(* CODESYS project HVAC Example Project.project

Project tree, tasks and I/O mapping:
  Device : CODESYS Control Win V3, 3S - Smart Software Solutions GmbH, order no. 305021, version 3.5.11.30
    application Application
      libraries: Standard, * (System); HVAC Library, 1.4.0.0 (Pfaender GmbH); HVAC Types Library, 1.0.0.0 (Pfaender GmbH); HVAC Visu Library, 1.2.0.0 (Pfaender GmbH); VisuDialogs, * (System); Util, * (System)
      task HIGH (cyclic, interval t#5ms, priority 1) calls AC_CALL_HIGH_START, AC_CALL_HIGH_END
      task LOW (cyclic, interval t#20ms, priority 10) calls AC_CALL_LOW_START, AC_CALL_LOW_END
      task TrendRecordingTask (cyclic, interval 100 ms, priority 31) calls VisuTrendStorageAccess.GlobalInstances.g_TrendRecordingManager.CyclicCall
      task MainTask (cyclic, interval t#20ms, priority 1) calls PRG, Main
      task AC_RMP_Task (cyclic, interval t#20ms, priority 30) calls AC_PRG_RMP
      task AlarmManagerTask (cyclic, interval 50 ms, priority 31) calls AlarmManager.Alarm_Prg
      task VISU_TASK (cyclic, interval 100 ms, priority 31) calls VisuElems.Visu_Prg
      Trend Recording Manager
        HC_1_Trend
      Visu/
        visualisation Header_Frame
        3_Settings/
          visualisation Settings_Start
          visualisation Settings_Persistence
          visualisation Settings_MANInfo
        2_Clock Settings/
          visualisation Clock_Settings_Start
          visualisation Clock_Holiday
          visualisation Clock_Public_Holiday
          visualisation Clock_SwitchTimeS
        1_Objects/
          HC_1/
            visualisation Settings_HC_1
            visualisation Heatcurve_HC_1
            visualisation Trend_HC_1
            visualisation Clock_HC_1
            visualisation Start_HC_1
          Room_1/
            visualisation Clock_Room_1
            visualisation Start_Room_1
          visualisation Objects_Start
          AHU_1/
            visualisation Start_AHU_1
            visualisation Clock_AHU_1
        0_Alarm/
          visualisation Alarm_Start
        4_Weather/
          visualisation Weather_Start
      visualisation Start
      program Main [CFC]
      text PersistenceConfig
      AC_Std/
        function AC_InitInternal [ST]
        global variables MODULE_INFOS
        function AC_OnlineChange [ST]
        program AC_CALL_LOW_END [ST]
        program AC_CALL_LOW_START [ST]
        global variables GVL_MODULE_TREE
        program AC_CALL_HIGH_END [ST]
        program AC_CALL_HIGH_START [ST]
        global variables GVL_PersistenceManager
        function AC_Init [ST]
      Alarm Configuration
        alarm class Warning (priority 30, acknowledge REP)
        alarm group AlarmGroup
            1 [Info]: Comparison Equal, ExpressionToCompare TRUE, Expression Main.xInfoTest - "Test Alarm Class Info"
            2 [Warning]: Comparison Equal, ExpressionToCompare TRUE, Expression Main.xWarningTest - "Test Alarm Class Warning"
            3 [Error]: Comparison Equal, ExpressionToCompare TRUE, Expression PRG.HC_1.Pump.xAlarm - "Heizkreis 1: Pumpe"
            4 [Error]: Comparison Equal, ExpressionToCompare TRUE, Expression PRG.HC_1.Pump.xAlarmFb - "Heizkreis 1: Pumpe Betriebsüberwachung"
            5 [Error]: Comparison Equal, ExpressionToCompare TRUE, Expression PRG.HC_1.TS_FT_ERR - "Heizkreis 1:  Vorlauftemperaturfühler Wert gestört"
            6 [Error]: Comparison Equal, ExpressionToCompare TRUE, Expression PRG.HC_1.TS_RT_ERR - "Heizkreis 1:  Rücklauftemperaturfühler Wert gestört"
            7 [Error]: Comparison Equal, ExpressionToCompare TRUE, Expression PRG.HC_1.Valve.xAlarm - "Heizkreis 1: Ventil"
            19 [Error]: Comparison Equal, ExpressionToCompare TRUE, Expression PRG.AHU_1.Fan.xAlarm - "RLT1: Abluftventilator"
            21 [Warning]: Comparison Equal, ExpressionToCompare FALSE, Expression PRG.AHU_1.BA_AUTO - "RLT1: Anlagenschalter auf Handbetrieb"
            10 [Warning]: Comparison NotEqual, ExpressionToCompare 0, Expression PRG.HC_1.Pump.eManModeB - "Heizkreis 1: Pumpe auf Handbetrieb (Software)"
            24 [Warning]: Comparison NotEqual, ExpressionToCompare 0, Expression PRG.AHU_1.Fan_AOO - "RLT1: Ventilator auf Handbetrieb (Hardware)"
            25 [Warning]: Comparison NotEqual, ExpressionToCompare 0, Expression PRG.AHU_1.OA_Damper_AOO - "RLT1: Außenluftklappe auf Handbetrieb (Hardware)"
            16 [Warning]: Comparison NotEqual, ExpressionToCompare 0, Expression PRG.Room_1.VEN_AOO - "Room 1: Ventil auf Handbetrieb (Hardware)"
            12 [Warning]: Comparison Equal, ExpressionToCompare FALSE, Expression PRG.HC_1.BA_AUTO - "Heizkreis 1: Anlagenwahlschalter auf Handbetrieb (Software)"
            22 [Warning]: Comparison NotEqual, ExpressionToCompare 0, Expression PRG.AHU_1.Damper_OutsideAir.eManModeB - "RLT1: Außenluftklappe auf Handbetrieb (Software)"
            11 [Warning]: Comparison NotEqual, ExpressionToCompare 0, Expression PRG.HC_1.Valve.eManModeN - "Heizkreis 1: Ventil auf Handbetrieb (Software)"
            13 [Error]: Comparison Equal, ExpressionToCompare TRUE, Expression PRG.Room_1.RBG_TF_RT_STO - "Room 1: Raumtemperaturfühler Wert gestört"
            23 [Warning]: Comparison NotEqual, ExpressionToCompare 0, Expression PRG.AHU_1.Fan.eManModeB - "RLT1: Ventilator auf Handbetrieb (Software)"
            17 [Warning]: Comparison NotEqual, ExpressionToCompare 0, Expression PRG.Room_1.VEN.eManModeB - "Room 1: Ventil auf Handbetrieb (Software)"
            8 [Warning]: Comparison NotEqual, ExpressionToCompare 0, Expression PRG.HC_1.Pump_AOO - "Heizkreis 1: Pumpe auf Handbetrieb (Hardware)"
            9 [Warning]: Comparison NotEqual, ExpressionToCompare 0, Expression PRG.HC_1.Valve_AO - "Heizkreis 1: Ventil auf Handbetrieb (Hardware)"
            14 [Error]: Comparison Equal, ExpressionToCompare TRUE, Expression PRG.Room_1.FROST - "Room 1: Frostgefahr"
            15 [Warning]: Comparison Equal, ExpressionToCompare FALSE, Expression PRG.Room_1.BA_AUTO - "Room 1: Anlagenschalter Betriebsmodus auf Handbetrieb"
            20 [Warning]: Comparison Equal, ExpressionToCompare TRUE, Expression PRG.AHU_1.FilterMonitoringB.xAlarm - "RLT1: Abluftfilter Wartung notwendig"
            18 [Error]: Comparison Equal, ExpressionToCompare TRUE, Expression PRG.AHU_1.Damper_OutsideAir.xAlarm - "RLT1: Außenluftklappe Störung"
            0 [Error]: Comparison Equal, ExpressionToCompare TRUE, Expression Main.xErrorTest - "Test Alarm Class Error"
        alarm class Error (priority 10, acknowledge REP_ACK)
        text list AlarmGroup
        alarm class Info (priority 100, acknowledge REP)
        AlarmStorage
      Macros and frames/
        Room_DE/
          visualisation Zone_F_Therm_Start
          function block Zone_F_Therm [CFC]
        HeatingCircuit/
          visualisation HeatCurve4P_DN
          function block HeatingCircuit_VenA [CFC]
          visualisation HeatingCircuit_VenA_Settings
          Pump_Frames/
            visualisation Pump_Button
            visualisation Pump_Parameter_Dialog
          Valve_Frames/
            visualisation ValveAnalog_Parameter_Dialog
            visualisation ValveAnalog_Button
          visualisation HeatingCircuit_VenA
        Clock/
          visualisation Holiday
          visualisation PublicHoliday
          visualisation SwitchTimeS
        Exhaust air system/
          visualisation ExhaustAir
          function block ExhaustAir [CFC]
      program PRG [CFC]
      AC_FBs/
        function block AC_PersistenceManager_HVAC_Parameter [ST]
        function block AC_PersistenceManager_HVAC_Counter [ST]
        function block AC_PersistenceManager [ST]
      AC_RMP/
        program AC_PRG_RMP [ST]
        global variables AC_RMP
  libraries: AC_Persistence, * (3S - Smart Software Solutions GmbH)
  5ce3da45-db07-42e7-a21c-a00fff4ed8f6|C:\Users\Lukas_Pfaender\Desktop\bilder codesys\Warnung_aktiv.gif
  5ce3da45-db07-42e7-a21c-a00fff4ed8f6|C:\Users\Lukas_Pfaender\Desktop\bilder codesys\Wartung.gif
  5ce3da45-db07-42e7-a21c-a00fff4ed8f6|C:\Users\Lukas_Pfaender\Desktop\bilder codesys\Alarm_aktiv.gif
  PersistenceManager
    Kanäle (pChannels)
      HVAC_Parameter
        Datenspeicher (itfDataStorage)
        ASCIIFileStorage
      HVAC_Counter
        Datenspeicher (itfDataStorage)
        ASCIIFileStorage
  text list GlobalTextList
  AC_GENERATOR_DATA
  5ce3da45-db07-42e7-a21c-a00fff4ed8f6|C:\Users\Lukas_Pfaender\Desktop\bilder codesys\Alarm_inaktiv.gif
  GlobalImagePool
  text list System
*)

// Device/Application/AC_Std/MODULE_INFOS
//Code generated by Application Composer.
//Modifying generated code is not recommended!
{attribute 'global_init_slot' := '40000'}
{attribute 'init_on_onlchange'}

VAR_GLOBAL
	{attribute 'init_on_onlchange'}
	AC_PERSIST_PersistenceManager_INFO: AC_PERSIST.AC.ModuleInfo := (pbyModuleType := ADR('AC_PERSIST.PersistenceManager'));
	{attribute 'init_on_onlchange'}
	AC_PERSIST_PersistenceChannel_INFO: AC_PERSIST.AC.ModuleInfo := (pbyModuleType := ADR('AC_PERSIST.PersistenceChannel'));
	{attribute 'init_on_onlchange'}
	AC_PERSIST_ASCIIFileStorage_INFO: AC_PERSIST.AC.ModuleInfo := (pbyModuleType := ADR('AC_PERSIST.ASCIIFileStorage'));
END_VAR

// Device/Application/AC_Std/GVL_MODULE_TREE
//Code generated by Application Composer.
//Modifying generated code is not recommended!

VAR_GLOBAL
	Module_Tree: AC_PERSIST.AC.ModuleTree;
	aNodes: ARRAY[0..5] OF AC_PERSIST.AC.MNode;
	AC_Environment: AC_PERSIST.AC.MEnv;
END_VAR

// Device/Application/AC_Std/GVL_PersistenceManager
//Code generated by Application Composer.
//Modifying generated code is not recommended!

VAR_GLOBAL
	PersistenceManager: AC_PersistenceManager;
END_VAR

// Device/Application/AC_RMP/AC_RMP
//Code generated by Application Composer.
//Modifying generated code is not recommended!
{attribute 'global_init_slot' := '60000'}
{attribute 'init_on_onlchange'}

VAR_GLOBAL
	{attribute 'init_on_onlchange'}
	AC_RMP_Service: AC_PERSIST.AC.RMPService := (uiLocalAppID:=9744, uiNumberOfConnections:=0, pSendConnection:=0, pReceiveConnection:=0);
END_VAR

// Device/Application/AC_Std/AC_CALL_HIGH_START
//Code generated by Application Composer.
//Modifying generated code is not recommended!
PROGRAM AC_CALL_HIGH_START

//Code generated by Application Composer.
//Modifying generated code is not recommended!
PersistenceManager.CallPrioHIGHStart() ;

END_PROGRAM

// Device/Application/AC_Std/AC_CALL_HIGH_END
//Code generated by Application Composer.
//Modifying generated code is not recommended!
PROGRAM AC_CALL_HIGH_END

//Code generated by Application Composer.
//Modifying generated code is not recommended!
PersistenceManager.CallPrioHIGHEnd() ;

END_PROGRAM

// Device/Application/AC_Std/AC_CALL_LOW_START
//Code generated by Application Composer.
//Modifying generated code is not recommended!
PROGRAM AC_CALL_LOW_START

//Code generated by Application Composer.
//Modifying generated code is not recommended!
PersistenceManager.CallPrioLOWStart() ;

END_PROGRAM

// Device/Application/AC_Std/AC_CALL_LOW_END
//Code generated by Application Composer.
//Modifying generated code is not recommended!
PROGRAM AC_CALL_LOW_END

//Code generated by Application Composer.
//Modifying generated code is not recommended!
PersistenceManager.CallPrioLOWEnd() ;

END_PROGRAM

// Device/Application/PRG
PROGRAM PRG
VAR
	
	GebVar: STRING;
	HC_1: HeatingCircuit_VenA;
	HC_1_Line1 : HVAC.EditString;
	
	Room_1 : Zone_F_Therm;
	Room_Line1: HVAC.EditString;
	Clock7d1Ch_Demo: HVAC.Clock7d1Ch;
	Clock7d2Ch_Demo: HVAC.Clock7d2Ch;
	Holiday_Demo: HVAC.Holiday;
	SwitchTimeS_Demo: HVAC.SwitchTimeS;
	PublicHoliday_Demo: HVAC.PublicHoliday;

	AHU_1_Line1: HVAC.EditString;
	AHU_1: ExhaustAir;
END_VAR

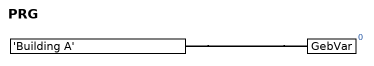
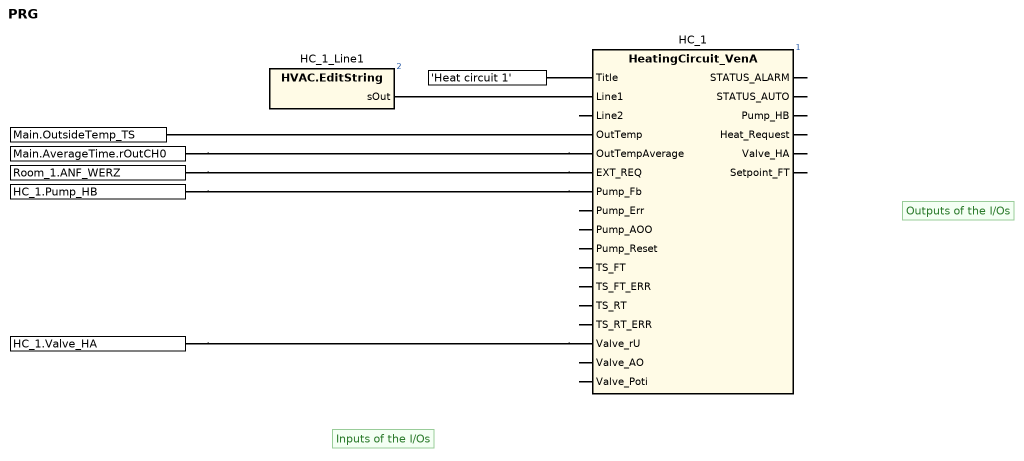
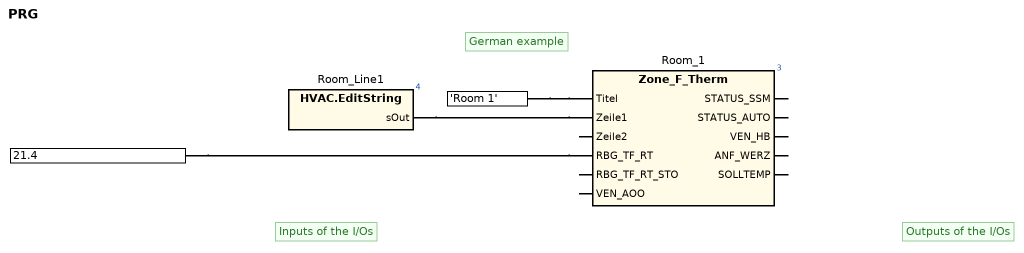
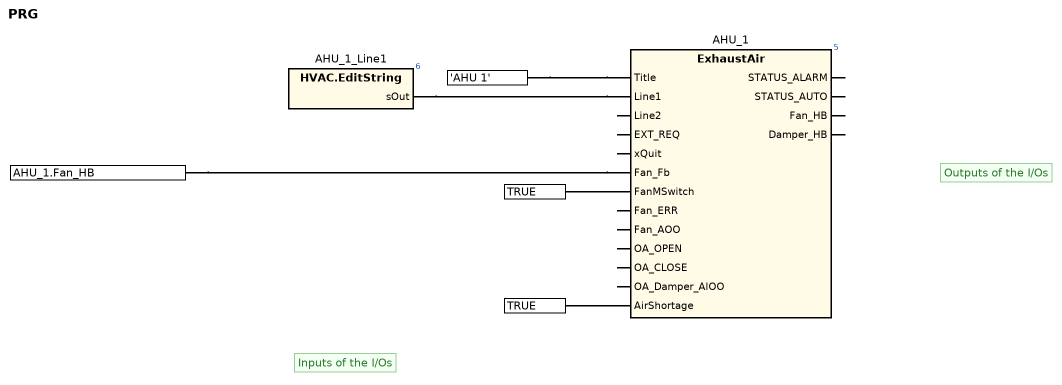
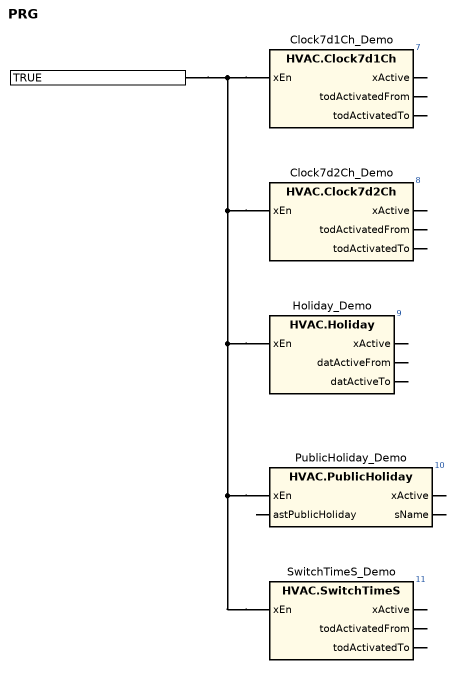
GebVar := 'Building A';
// Outputs of the I/Os
HC_1(
    Title := 'Heat circuit 1',
    Line1 := HC_1_Line1.sOut,
    OutTemp := Main.OutsideTemp_TS,
    OutTempAverage := Main.AverageTime.rOutCH0,
    EXT_REQ := Room_1.ANF_WERZ,
    Pump_Fb := HC_1.Pump_HB,
    Valve_rU := HC_1.Valve_HA); // HeatingCircuit_VenA
// Inputs of the I/Os
// parameter HC_1_Line1.sSetPoint := 'Zone 2+3'
HC_1_Line1(); // HVAC.EditString
// German example
// Outputs of the I/Os
Room_1(Titel := 'Room 1', Zeile1 := Room_Line1.sOut, RBG_TF_RT := 21.4); // Zone_F_Therm
// Inputs of the I/Os
// parameter Room_Line1.sSetPoint := 'Mr. John Doe'
Room_Line1(); // HVAC.EditString
// Outputs of the I/Os
AHU_1(
    Title := 'AHU 1',
    Line1 := AHU_1_Line1.sOut,
    Fan_Fb := AHU_1.Fan_HB,
    FanMSwitch := TRUE,
    AirShortage := TRUE); // ExhaustAir
// Inputs of the I/Os
// parameter AHU_1_Line1.sSetPoint := 'Air handling unit - exhaust air'
AHU_1_Line1(); // HVAC.EditString
Clock7d1Ch_Demo(xEn := TRUE); // HVAC.Clock7d1Ch
Clock7d2Ch_Demo(xEn := TRUE); // HVAC.Clock7d2Ch
Holiday_Demo(xEn := TRUE); // HVAC.Holiday
PublicHoliday_Demo(xEn := TRUE); // HVAC.PublicHoliday
SwitchTimeS_Demo(xEn := TRUE); // HVAC.SwitchTimeS

END_PROGRAM

// Device/Application/Main
PROGRAM Main
VAR

	TimeRead: HVAC.TimeRead;
	StartDelay: HVAC.StartDelay;
	AverageTime: HVAC.AverageTime;
	AlarmCounter: HVAC.AlarmCounter;
	Alarmgroup : UDINT := Alm_AlarmConfiguration_Alarmgroup_InternalIDs.ID_AlarmGroup;
	
	ManInfo: HVAC.ManInfo;
	ManBin_Test1: HVAC.ManBin;
	ManNum_Test1: HVAC.ManNum;
	OutsideTemp_TS: REAL := 18.5;  // Outside temperature sensor dummy. normaly analog input.

	Alarm_blink: BLINK;
	xAlarme_blinker: BOOL;
	
	xErrorTest: BOOL;
	xInfoTest  : BOOL;
	xWarningTest:BOOL;
	AlarmCounter_Warning: HVAC.AlarmCounter;
	
	OutsideTemp_TS_ERR: BOOL;						// Störung Außentemperaturfühler // Error outside temperature sensor
	checkLicense: HVAC.checkLicense;
	Outside_Temp_MAN: HVAC.ManNum;
END_VAR

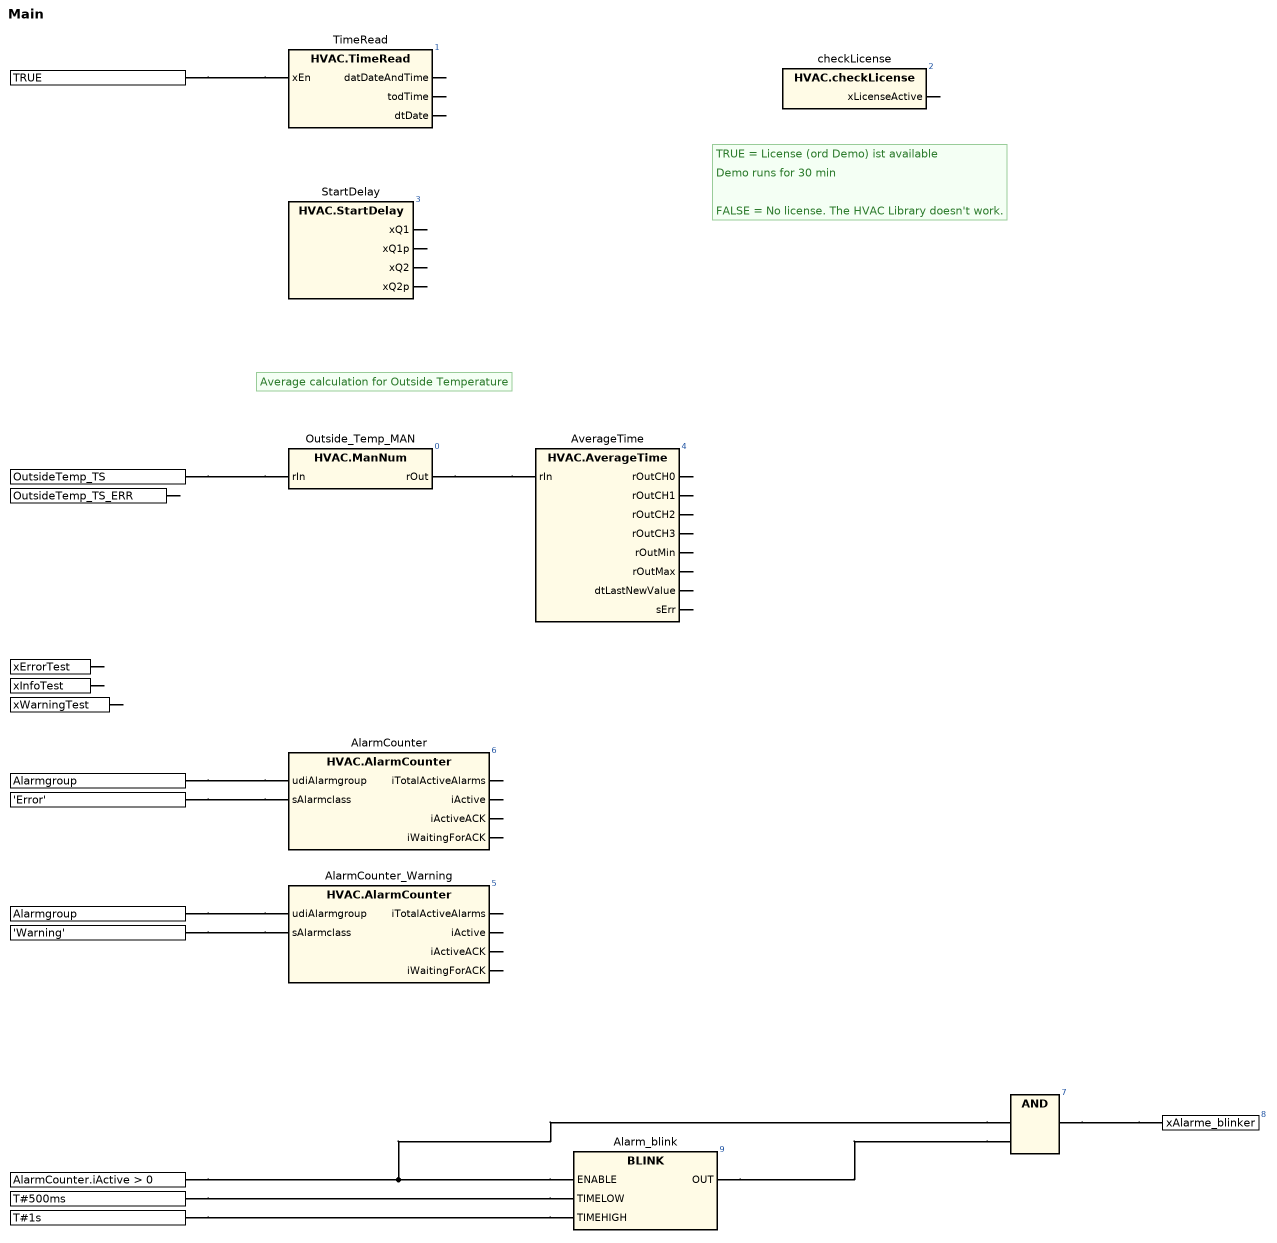
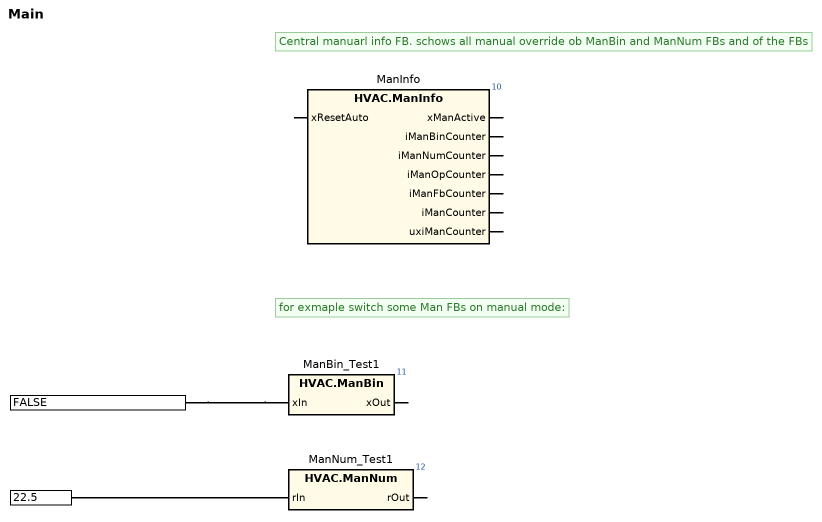
// Average calculation for Outside Temperature
Outside_Temp_MAN(rIn := OutsideTemp_TS); // HVAC.ManNum
TimeRead(xEn := TRUE); // HVAC.TimeRead
checkLicense(); // HVAC.checkLicense
// TRUE = License (ord Demo) ist available
// Demo runs for 30 min
//
// FALSE = No license. The HVAC Library doesn't work.
StartDelay(); // HVAC.StartDelay
AverageTime(rIn := Outside_Temp_MAN.rOut); // HVAC.AverageTime
AlarmCounter_Warning(udiAlarmgroup := Alarmgroup, sAlarmclass := 'Warning'); // HVAC.AlarmCounter
AlarmCounter(udiAlarmgroup := Alarmgroup, sAlarmclass := 'Error'); // HVAC.AlarmCounter
xAlarme_blinker := (AlarmCounter.iActive > 0) AND Alarm_blink.OUT;
Alarm_blink(ENABLE := AlarmCounter.iActive > 0, TIMELOW := T#500ms, TIMEHIGH := T#1s); // BLINK
// Central manuarl info FB. schows all manual override ob ManBin and ManNum FBs and of the FBs
ManInfo(); // HVAC.ManInfo
// for exmaple switch some Man FBs on manual mode:
ManBin_Test1(xIn := FALSE); // HVAC.ManBin
ManNum_Test1(rIn := 22.5); // HVAC.ManNum
// OutsideTemp_TS_ERR: input not connected
// xInfoTest: input not connected
// xWarningTest: input not connected
// xErrorTest: input not connected

END_PROGRAM

// Device/Application/Macros and frames/HeatingCircuit/HeatingCircuit_VenA
FUNCTION_BLOCK HeatingCircuit_VenA
VAR_INPUT
	Title						: STRING; 						// Name des Heizkreises  // Name of the heating circuit
	Line1						: STRING; 						// Zeile eins der Kachel // Description line 1
	Line2						: STRING; 						// Zeile zwei der Kachel // Description Line 1
	OutTemp						: REAL;							// Aussentemperaturfühler  // Outside temperature sensor
	OutTempAverage				: REAL;							// Aussentemperaturdurchschnitt // Outside temperature average
	EXT_REQ						: BOOL := FALSE;				// Externe Anforderung (Verbraucher) // External Requirement (Consumer)
	Pump_Fb						: BOOL; 						// Betrieb Umwälzpumpe // Feedback pump
	Pump_Err					: BOOL;							// Störung von Umwälzpumpe  // Alarm pump
	Pump_AOO					: HVACTypes.eManBin;			// Automatik Umwälzpumpe // pump hardware manual override(A)uto (O)ff (O)n
	Pump_Reset					: BOOL := FALSE;				// Reseteingang Störung Überwachung Betrieb  // Reset input for deedback control
	TS_FT						: REAL;							// Vorlauftemperatur // Temperature sensor flow temperature
	TS_FT_ERR					: BOOL;							// Störung Vorlauftemperaturfühler // Temperature sensor flow temperature ERROR
	TS_RT						: REAL;							// Rücklauftemperatur // Temperature sensor return temperature
	TS_RT_ERR					: BOOL;							// Störung Rücklauftemperaturfühler // Temperature sensor return temperature ERROR
	Valve_rU					: REAL;							// Rückführung Ventil  // Return Valve
	Valve_AO					: HVACTypes.eManNum;							// Automatik Ventil  //  Valve hardware manual override (A)uto (On)
	Valve_Poti					: REAL;							// Analogübersteuerung Poti // manual override potentiometer value
END_VAR

VAR_OUTPUT
	STATUS_ALARM					: BOOL;							// Sammelstörmeldung // Central Fault (Error)
	STATUS_AUTO					: BOOL;							// Statusmeldung: 0=Hand 1=Auto // Central Automatic message FALSE = manual TRUE = Auto
	Pump_HB						: BOOL;							// Ausgang Umwälzpumpe  // Output pump binary
	Heat_Request				: BOOL;							// Anforderung Wärmeerzeugung  // Heat request
	Valve_HA					: REAL;							// Ausgang Ventil // Output valve analog
	Setpoint_FT					: REAL;							// Vorlaufsolltemperatur  // Setpoint flow temperature
END_VAR
VAR
	OS							: hvac.OpModeSelect;			// Anlagen Wahlschalter // Operation mode Select
	BA_AUTO						: BOOL;							// Betriebsart Auto // Operation mode automatic
	BA_HAND0					: BOOL;							// Betriebsart HAND - Nachtbetrieb  // Operation mode: manual - night operation
	BA_HAND1					: BOOL;							// Betriebsart HAND - Tagbetrieb // Operation mode: manual - day operation
	R_OutTemp					: BOOL;							// Freigabe über Aussentemperatur  // Release via outside temperature
	R_OutTemp_MAN				: hvac.ManBin;					// Manuell Baustein für die Freigabe der Außentemperatur  // Manual function block for outside temperature release
	R_OutTemp_SR				: SR;							// Flipflop Freigabe Heizbetrieb  // Release flipflop for heating operation
	R_OutTemp_TON				: TON;							
	R_OutTemp_TOF				: TOF;
	HEAT						: BOOL;							// Heizbetrieb  // Heating operation
	HC							: hvac.HeatCurve4P_DN;			// Heizkurve // haeting curve
	MODE						: BOOL;							// Modus: FALSE=Nachtbetrieb TRUE=Tagbetrieb // Mode: FALSE=night operation TRUE=day operation
	Reg2P_HZ_AKT				: hvac.Control2P;				// Zweipunktregler Heizen aktuell  // Control two point heating mode actual
	Reg2P_HZ_DURCH				: hvac.Control2P;				// Zweipunktregler Heizen Durchschnitt //  Control two point heating mode average
	Reg2P_WINTER				: hvac.Control2P;				// Zweipunktregler Heizen Wintermodus // Control two point heating operation winter
	ConPI_FT					: hvac.ControlPI;				// PI Regler für Vorlauftemperaturregelung	// Control PI for flow temperature regulation
	Setpoint_FT_MAN				: hvac.ManNum;					// Handübersteuerung Soll Vorlauftemperatur // Manual override for setpoint flow temperature
	Setpoint_Heat_Aver				: hvac.Edit;					// Sollwert: Freigabe Heizbetrieb bei AT-Durch < // Setpoint: Release heating operation at outside temperature average <
	Setpoint_Heat_Act			: hvac.Edit;					// Sollwert: Freigabe Heizbetrieb bei Aussentemperatur < // Setpoint: Release heating operation at actual outside temperature <
	Setpoint_WINTER				: hvac.Edit;					// Sollwert: Freigabe Winterbetrieb bei AT-Durch < // Setpoint release winter operation at outside temperature average <
	STATUS_ERR_MAN				: hvac.ManBin;					// Handübersteuerung Sammelstörmeldung  // Manual override central error
	STATUS_AUTO_MAN				: hvac.ManBin;					// Handübersteuerung Automatikmeldung // Manual override central automatic notification
	Clock						: HVAC.Clock7d1Ch;				// Einkanal Wochenuhr  // One channel week clock
	Pump						: hvac.Pump;					// Umwälzpumpe  // Circuit  pump
	Clock_Channel				: BOOL;							// Uhrkanal // Clock Channel
	Valve_ERR					: BOOL;							// Störung Ventil //Valve Alarm
	WINTER						: BOOL;							// Winterbetrieb //Winter operation
	Valve						: hvac.ValveAnalog;
END_VAR
VAR // added by the converter: edge detectors and wires of the graphical bodies
    _w1, _w2, _w3, _w4, _w5, _w6, _w7 : ANY;
END_VAR

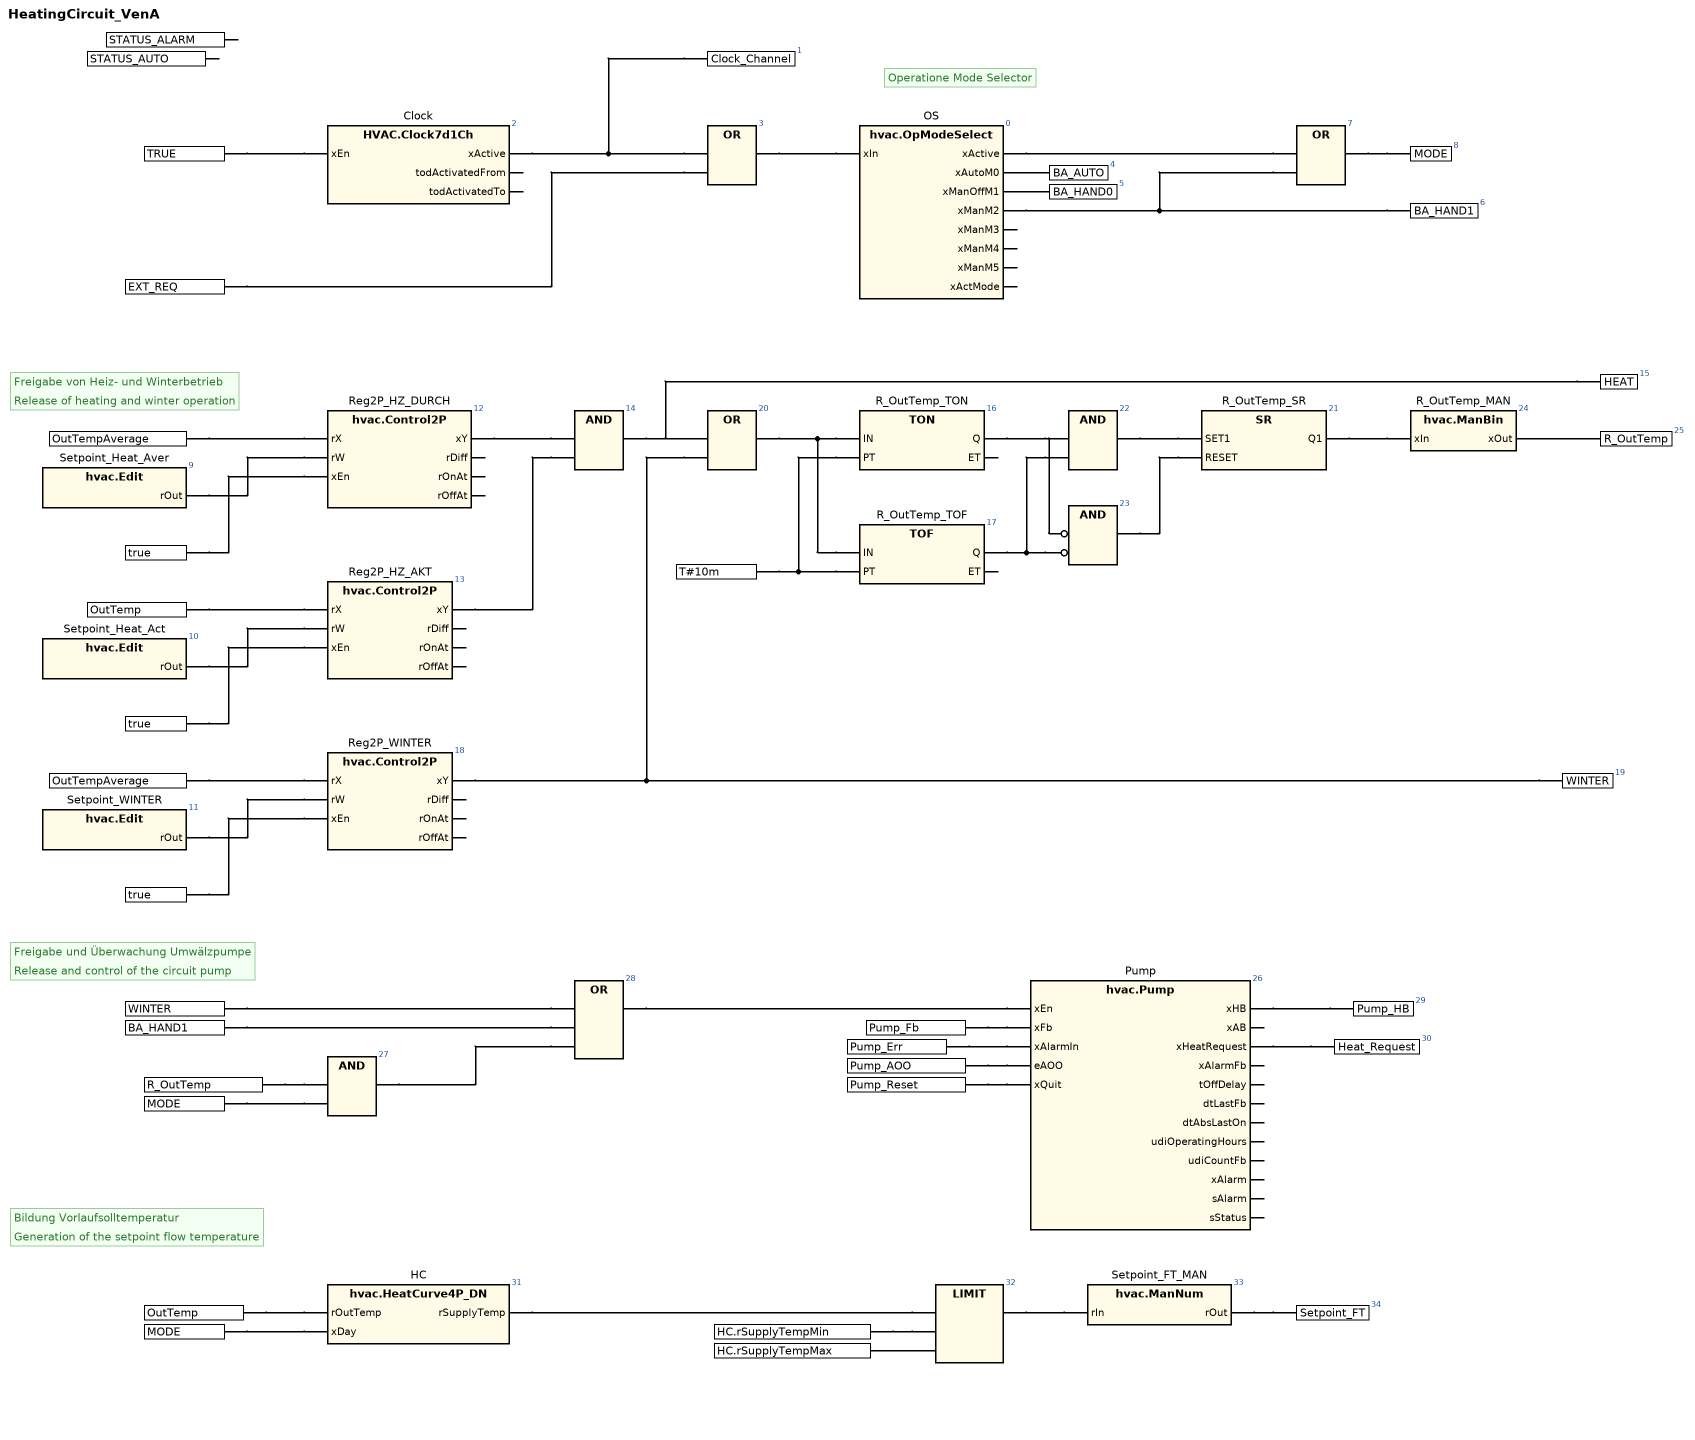
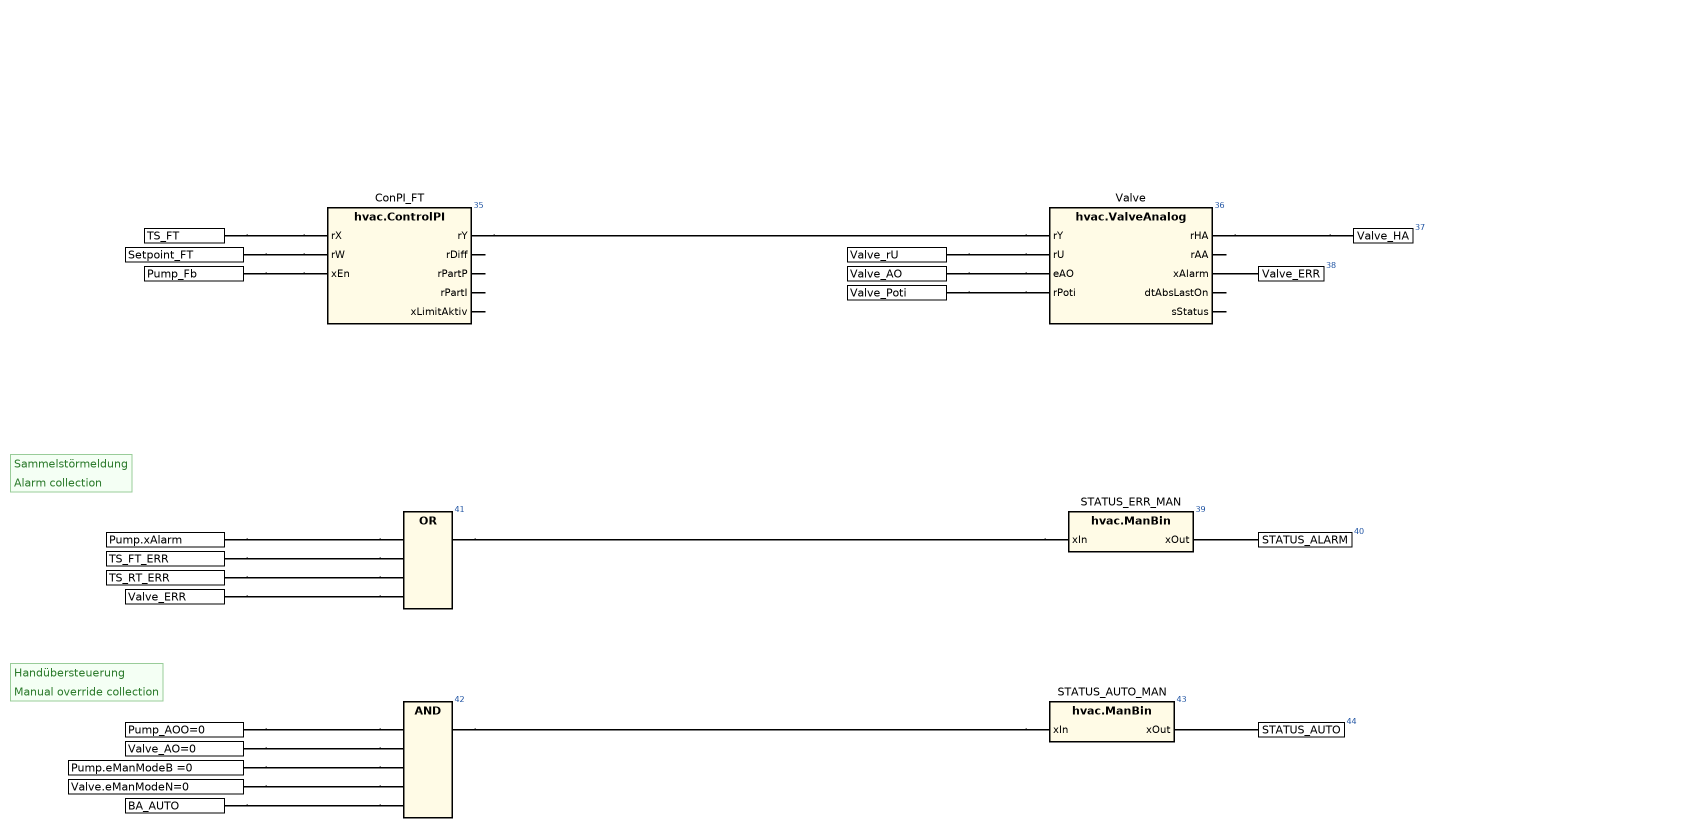
// note: 115 stored wires end on pins the file does not list and are not shown
// Operatione Mode Selector
// parameter OS.sTitleM2 := 'Manual On'
// parameter OS.sTitleM1 := 'Manual Off'
// parameter OS.sTitleM0 := 'Automatic'
// parameter OS.sTitle := 'Operation Mode'
// parameter OS.eMaxMode := HVAC.eOpMode.Mode2
OS(xIn := _w1); // hvac.OpModeSelect
Clock_Channel := Clock.xActive;
// parameter Clock.todSunTo := tod#00:00:00
// parameter Clock.todSunFrom := tod#00:00:00
// parameter Clock.todFriTo := tod#23:59:00
// parameter Clock.todFriFrom := tod#23:59:00
Clock(xEn := TRUE); // HVAC.Clock7d1Ch
_w1 := Clock.xActive OR EXT_REQ;
BA_AUTO := OS.xAutoM0;
BA_HAND0 := OS.xManOffM1;
BA_HAND1 := OS.xManM2;
MODE := OS.xActive OR OS.xManM2;
// Freigabe von Heiz- und Winterbetrieb
// Release of heating and winter operation
// parameter Setpoint_Heat_Aver.rSetPoint := 22
Setpoint_Heat_Aver(); // hvac.Edit
// parameter Setpoint_Heat_Act.rSetPoint := 20
Setpoint_Heat_Act(); // hvac.Edit
// parameter Setpoint_WINTER.rSetPoint := 8
Setpoint_WINTER(); // hvac.Edit
// parameter Reg2P_HZ_DURCH.rSwitchOnPoint := 
// parameter Reg2P_HZ_DURCH.rSwitchOffPoint := 
Reg2P_HZ_DURCH(rX := OutTempAverage, rW := Setpoint_Heat_Aver.rOut, xEn := true); // hvac.Control2P
Reg2P_HZ_AKT(rX := OutTemp, rW := Setpoint_Heat_Act.rOut, xEn := true); // hvac.Control2P
_w2 := Reg2P_HZ_DURCH.xY AND Reg2P_HZ_AKT.xY;
HEAT := _w2;
R_OutTemp_TON(IN := _w3, PT := T#10m); // TON
R_OutTemp_TOF(IN := _w3, PT := T#10m); // TOF
Reg2P_WINTER(rX := OutTempAverage, rW := Setpoint_WINTER.rOut, xEn := true); // hvac.Control2P
WINTER := Reg2P_WINTER.xY;
_w3 := _w2 OR Reg2P_WINTER.xY;
R_OutTemp_SR(SET1 := _w4, RESET := _w5); // SR
_w4 := R_OutTemp_TON.Q AND R_OutTemp_TOF.Q;
_w5 := NOT R_OutTemp_TON.Q AND NOT R_OutTemp_TOF.Q;
R_OutTemp_MAN(xIn := R_OutTemp_SR.Q1); // hvac.ManBin
R_OutTemp := R_OutTemp_MAN.xOut;
// parameter Pump.udiFbControlTime := 20
Pump(xEn := _w6, xFb := Pump_Fb, xAlarmIn := Pump_Err, eAOO := Pump_AOO, xQuit := Pump_Reset); // hvac.Pump
// Freigabe und Überwachung Umwälzpumpe
// Release and control of the circuit pump
_w6 := WINTER OR BA_HAND1 OR R_OutTemp AND MODE;
Pump_HB := Pump.xHB;
Heat_Request := Pump.xHeatRequest;
// Bildung Vorlaufsolltemperatur
// Generation of the setpoint flow temperature
HC(rOutTemp := OutTemp, xDay := MODE); // hvac.HeatCurve4P_DN
Setpoint_FT_MAN(rIn := LIMIT(HC.rSupplyTemp, HC.rSupplyTempMin, HC.rSupplyTempMax)); // hvac.ManNum
Setpoint_FT := Setpoint_FT_MAN.rOut;
ConPI_FT(rX := TS_FT, rW := Setpoint_FT, xEn := Pump_Fb); // hvac.ControlPI
Valve(rY := ConPI_FT.rY, rU := Valve_rU, eAO := Valve_AO, rPoti := Valve_Poti); // hvac.ValveAnalog
Valve_HA := Valve.rHA;
Valve_ERR := Valve.xAlarm;
STATUS_ERR_MAN(xIn := _w7); // hvac.ManBin
STATUS_ALARM := STATUS_ERR_MAN.xOut;
// Sammelstörmeldung
// Alarm collection
_w7 := Pump.xAlarm OR TS_FT_ERR OR TS_RT_ERR OR Valve_ERR;
// Handübersteuerung
// Manual override collection
STATUS_AUTO_MAN(xIn := (Pump_AOO=0) AND (Valve_AO=0) AND (Pump.eManModeB =0) AND (Valve.eManModeN=0) AND BA_AUTO); // hvac.ManBin
STATUS_AUTO := STATUS_AUTO_MAN.xOut;
// STATUS_ALARM: input not connected
// STATUS_AUTO: input not connected

END_FUNCTION_BLOCK

// Device/Application/Macros and frames/Room_DE/Zone_F_Therm
FUNCTION_BLOCK Zone_F_Therm // Zone mit Temperaturfühler und thermischen Heizkörperventil - GERMAN EXAMPLE
VAR_INPUT
	Titel						: STRING; 						// Name der Zone
	Zeile1						: STRING; 						// Zeile eins der Kachel
	Zeile2						: STRING; 						// Zeile zwei der Kachel
	RBG_TF_RT					: REAL; 						// Raum Bediengerät Raumtemperatur
	RBG_TF_RT_STO				: BOOL; 						// Störung Raumtemperaturfühler
	VEN_AOO						: HVACTYPES.eManBin; 			// Automatik Ventil Auto, Off, On
	Lichttaster					: BOOL;							// Lichttaster // Light switch
	JAL_AUF						: BOOL;							// Jalousietaster AUF // Shade Up
	JAL_AB						: BOOL;							// Jalousietaster AB // Shade Down
END_VAR	
VAR_OUTPUT
	STATUS_SSM					: BOOL;							// Sammelstörmeldung
	STATUS_AUTO					: BOOL; 						// Statusmeldung: 0=Hand 1=Auto
	VEN_HB						: BOOL; 						// Ausgang Ventil
	Licht_HB					: BOOL;							// Ausgang Licht
	JAL_AUF_HB					: BOOL;							// Ausgang Jalousie AUF  // Output shade up
	JAL_ZU_HB					: BOOL;							// Ausgang Jalousie AB	// Output shade down
	ANF_WERZ					: BOOL;							// Anforderung Wärmeerzeugung
	SOLLTEMP					: REAL; 						// Solltemperatur

END_VAR
VAR
	AS							: HVAC.OpModeSelect;
	BA_AUTO						: BOOL;							// Betriebsart Auto
	BA_HAND0					: BOOL;							// Betriebsart HAND - Nachtbetrieb
	BA_HAND1					: BOOL;							// Betriebsart HAND - Tagbetrieb
	FROST						: BOOL; 						// Raumtemperatur ist zu niedrig --> Frostgefahr
	MODUS						: BOOL;							// Modus: 0=Nachtbetrieb 1=Tagbetrieb
	Reg2P_Frost					: HVAC.Control2P; 				// 2P-Regler Frostüberwachung im Raum
	Reg2P_RT					: HVAC.Control2P;				// 2P-Regler Raumtemperatur
	SOLLTEMP_MAN				: HVAC.ManNum;
	SOLLW_FROST					: HVAC.Edit;					// Solltemperatur Frostüberwachung
	SOLLW_NACHT					: hvac.Edit; 					// Solltemperatur Nachtbetrieb
	SOLLW_TAG					: hvac.Edit; 					// Solltemperatur Tagbetrieb
	STATUS_AUTO_MAN				: HVAC.ManBin;
	STATUS_SSM_MAN				: HVAC.ManBin;
	UHRKANAL					: BOOL;							// Uhrkanal
	VEN							: HVAC.ValveTherm;	
	Clock						: HVAC.Clock7d2Ch;
	VisuPoti: HVAC.EditPoti;
	LightButton: HVAC.ButtonToggle;
	Light_Man: HVAC.ManBin;
	Shade: HVAC.Shade;
	JAL_AUF_MAN: HVAC.ManBin;
	JAL_ZU_MAN: HVAC.ManBin;
	Lichttaster_Visu: BOOL;
	JAL_AUF_VISU: BOOL;
	JAL_AB_VISU: BOOL;
END_VAR
VAR // added by the converter: edge detectors and wires of the graphical bodies
    _w1 : BOOL;
    _w2, _w3, _w4, _w5, _w6, _w7, _w8 : ANY;
END_VAR

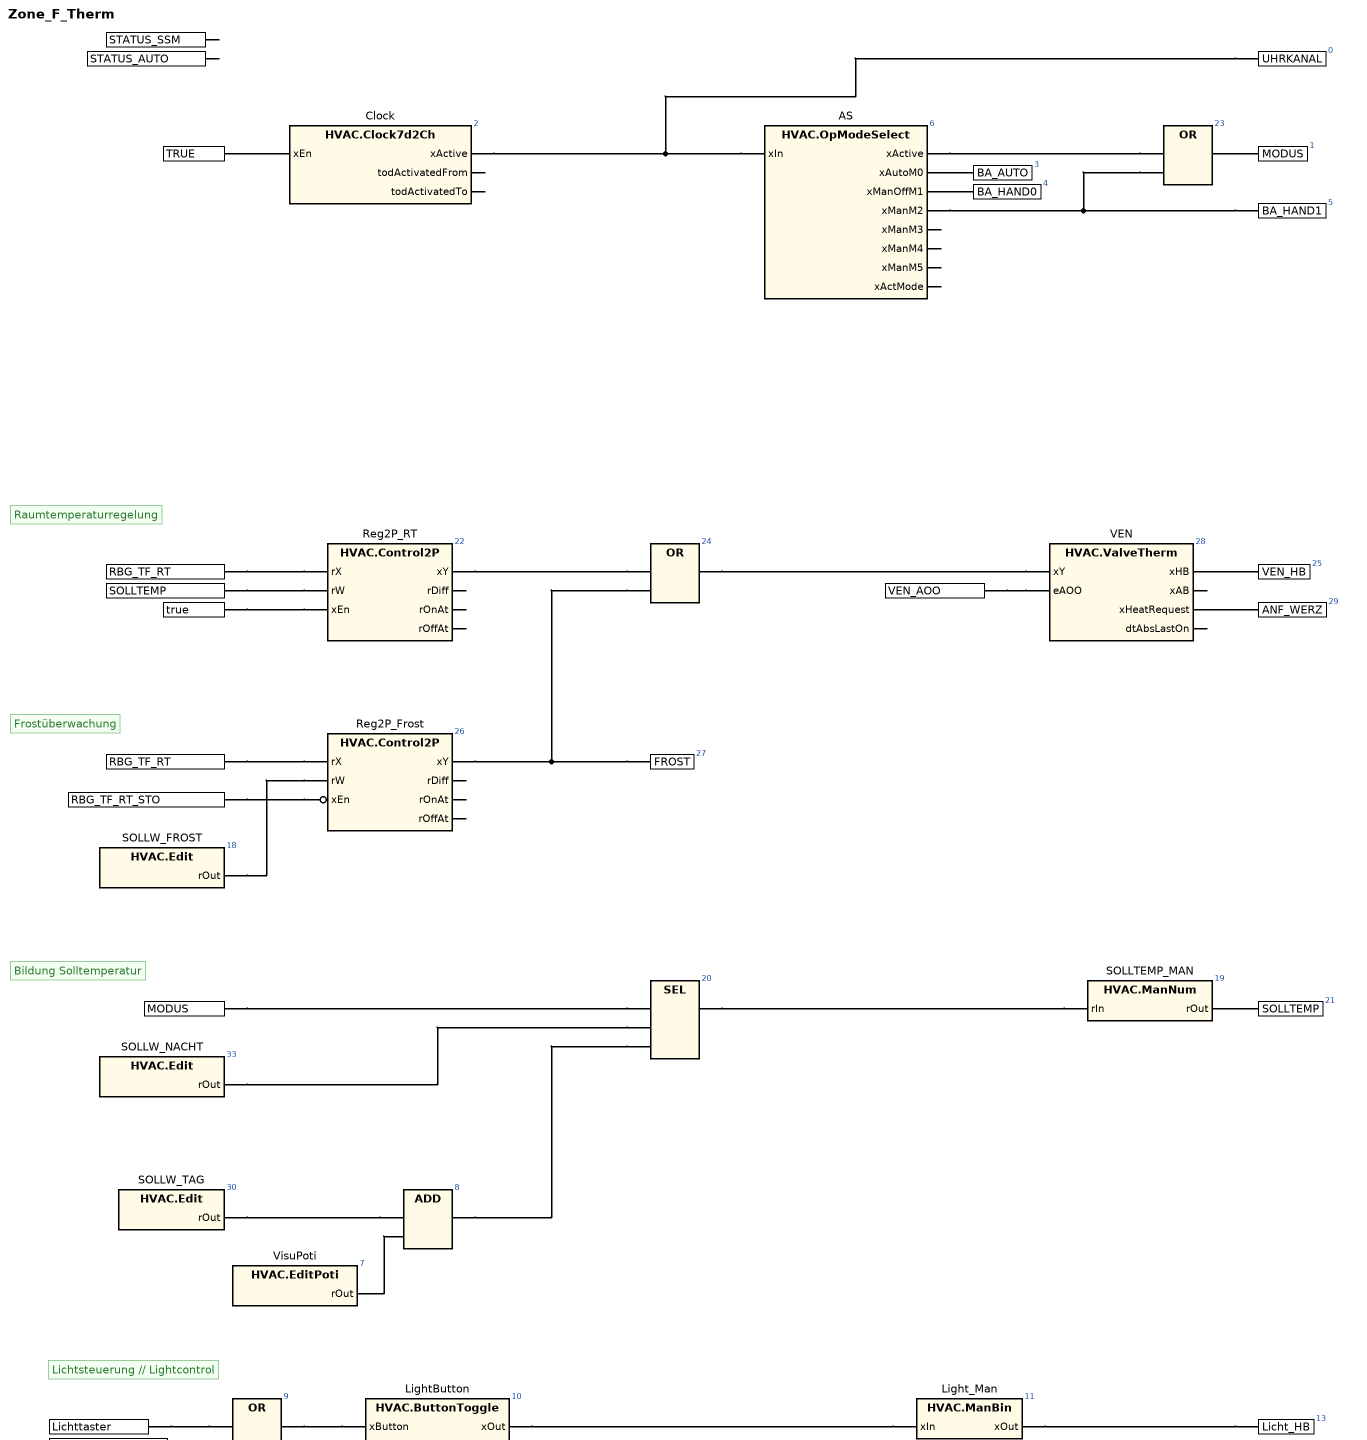
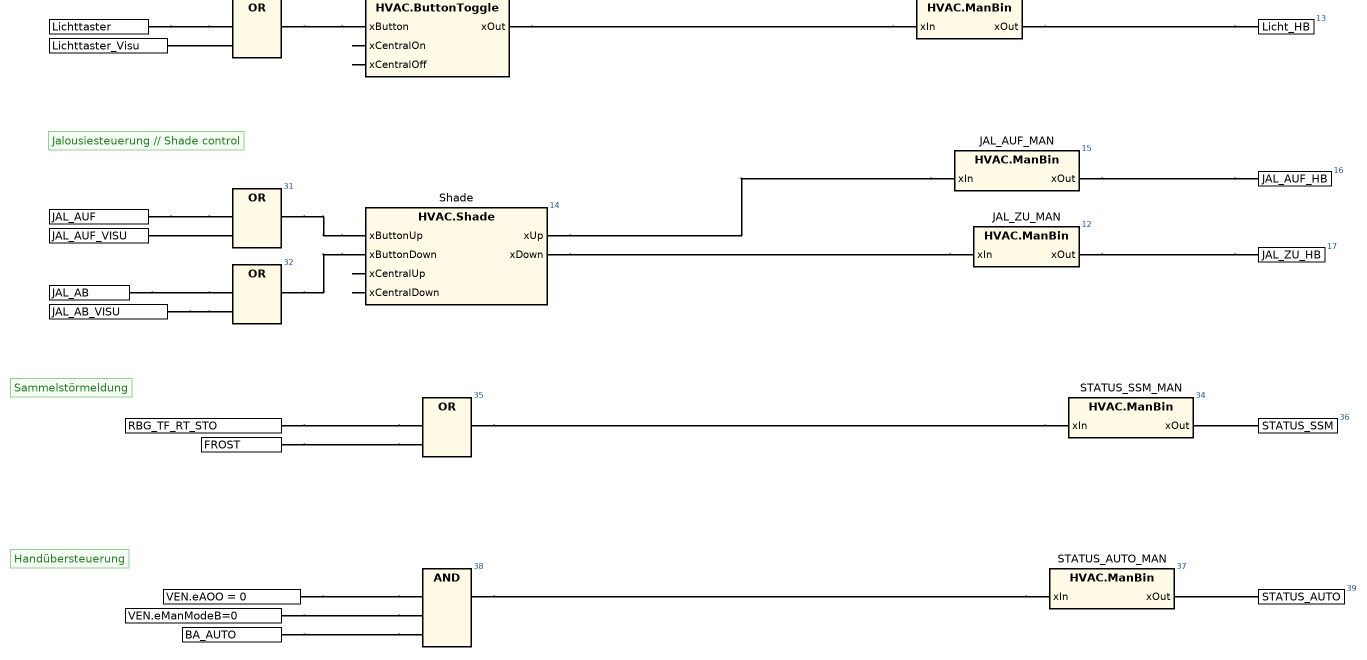
// note: 10 stored wires end on pins the file does not list and are not shown
UHRKANAL := Clock.xActive;
MODUS := _w1;
Clock(xEn := TRUE); // HVAC.Clock7d2Ch
BA_AUTO := AS.xAutoM0;
BA_HAND0 := AS.xManOffM1;
BA_HAND1 := AS.xManM2;
// parameter AS.sTitleM2 := 'Hand Ein - Tag'
// parameter AS.eMaxMode := HVAC.eOpMode.Mode2
AS(xIn := Clock.xActive); // HVAC.OpModeSelect
// parameter VisuPoti.rSetPointMin := -2
// parameter VisuPoti.rSetPointMax := 2
VisuPoti(); // HVAC.EditPoti
_w2 := SOLLW_TAG.rOut + VisuPoti.rOut;
// Lichtsteuerung // Lightcontrol
LightButton(xButton := Lichttaster OR Lichttaster_Visu); // HVAC.ButtonToggle
Light_Man(xIn := LightButton.xOut); // HVAC.ManBin
JAL_ZU_MAN(xIn := Shade.xDown); // HVAC.ManBin
Licht_HB := Light_Man.xOut;
Shade(xButtonUp := _w3, xButtonDown := _w4); // HVAC.Shade
JAL_AUF_MAN(xIn := Shade.xUp); // HVAC.ManBin
JAL_AUF_HB := JAL_AUF_MAN.xOut;
JAL_ZU_HB := JAL_ZU_MAN.xOut;
// Frostüberwachung
// parameter SOLLW_FROST.rSetPoint := 6
SOLLW_FROST(); // HVAC.Edit
SOLLTEMP_MAN(rIn := _w5); // HVAC.ManNum
_w5 := SEL(MODUS, SOLLW_NACHT.rOut, _w2);
SOLLTEMP := SOLLTEMP_MAN.rOut;
// Raumtemperaturregelung
// parameter Reg2P_RT.rSwitchOnPoint := -0.2
// parameter Reg2P_RT.rSwitchOffPoint := 0.2
Reg2P_RT(rX := RBG_TF_RT, rW := SOLLTEMP, xEn := true); // HVAC.Control2P
_w1 := AS.xActive OR AS.xManM2;
_w6 := Reg2P_RT.xY OR Reg2P_Frost.xY;
VEN_HB := VEN.xHB;
Reg2P_Frost(rX := RBG_TF_RT, rW := SOLLW_FROST.rOut, xEn := NOT RBG_TF_RT_STO); // HVAC.Control2P
FROST := Reg2P_Frost.xY;
VEN(xY := _w6, eAOO := VEN_AOO); // HVAC.ValveTherm
ANF_WERZ := VEN.xHeatRequest;
// parameter SOLLW_TAG.rSetPoint := 21
SOLLW_TAG(); // HVAC.Edit
// Jalousiesteuerung // Shade control
_w3 := JAL_AUF OR JAL_AUF_VISU;
_w4 := JAL_AB OR JAL_AB_VISU;
// Bildung Solltemperatur
// parameter SOLLW_NACHT.rSetPoint := 18
SOLLW_NACHT(); // HVAC.Edit
STATUS_SSM_MAN(xIn := _w7); // HVAC.ManBin
// Sammelstörmeldung
_w7 := RBG_TF_RT_STO OR FROST;
STATUS_SSM := STATUS_SSM_MAN.xOut;
STATUS_AUTO_MAN(xIn := _w8); // HVAC.ManBin
// Handübersteuerung
_w8 := (VEN.eAOO = 0) AND (VEN.eManModeB=0) AND BA_AUTO;
STATUS_AUTO := STATUS_AUTO_MAN.xOut;
// STATUS_SSM: input not connected
// STATUS_AUTO: input not connected

END_FUNCTION_BLOCK

// Device/Application/Macros and frames/Exhaust air system/ExhaustAir
FUNCTION_BLOCK ExhaustAir // AHU: Air Handling Unit for exhaust air
VAR_INPUT
	Title						: STRING; 						// Name des Heizkreises  // Name of the heating circuit
	Line1						: STRING; 						// Zeile eins der Kachel // Description line 1
	Line2						: STRING; 						// Zeile zwei der Kachel // Description Line 1
	EXT_REQ						: BOOL := FALSE;				// Externe Anforderung (Verbraucher) // External Requirement (Consumer)
	xQuit						: BOOL;							// Störung Entsperren // Quit Error
	Fan_Fb						: BOOL;							// Fan feedback
	FanMSwitch					: BOOL;							// Motor switch fan
	Fan_ERR						: BOOL;							// Fan Error
	Fan_AOO						: HVACTypes.eManBin;			// Automatikmeldugn Ventilator  //  Fan hardware manual override (A)uto (On) (O)ff
	OA_OPEN						: BOOL;							// Outside air damper OPEN feedback
	OA_CLOSE					: BOOL;							// Outside air damper CLOSE feedback
	OA_Damper_AOO				: HVACTypes.eManBin;			// Automatikmeldung Klappe  //  Damper hardware manual override (A)uto (On) (O)ff
	AirShortage					: BOOL;							// Differenzdruckschalter für Luftmangel // AirShortage
	Filter						: BOOL;							// Filter monitoring difference pressure binary
END_VAR

VAR_OUTPUT
	STATUS_ALARM				: BOOL;							// Sammelstörmeldung // Central Fault (Error)
	STATUS_AUTO					: BOOL;							// Statusmeldung: 0=Hand 1=Auto // Central Automatic message FALSE = manual TRUE = Auto
	Fan_HB						: BOOL;							// Fan output binary
	Damper_HB					: BOOL;							// Output damper binary
END_VAR
VAR
	OS							: hvac.OpModeSelect;			// Anlagen Wahlschalter // Operation mode Select
	BA_AUTO						: BOOL;							// Betriebsart Auto // Operation mode automatic
	BA_HAND0					: BOOL;							// Betriebsart HAND - Nachtbetrieb  // Operation mode: manual - night operation
	BA_HAND1					: BOOL;							// Betriebsart HAND - Tagbetrieb // Operation mode: manual - day operation
	Clock						: HVAC.Clock7d1Ch;				// Einkanal Wochenuhr  // One channel week clock
	Clock_Channel				: BOOL;							// Uhrkanal // Clock Channel
	Mode						: BOOL;							// Modus: FALSE=Nachtbetrieb TRUE=Tagbetrieb // Mode: FALSE=night operation TRUE=day operation
	Fan							: HVAC.Fan1Speed;
	Damper_OutsideAir			: HVAC.Damper2P;
	STATUS_ERR_MAN				: HVAC.ManBin;
	STATUS_AUTO_MAN				: HVAC.ManBin;
	FilterMonitoringB: HVAC.FilterMonitoringB;
END_VAR
VAR // added by the converter: edge detectors and wires of the graphical bodies
    _w1, _w2, _w3 : ANY;
END_VAR

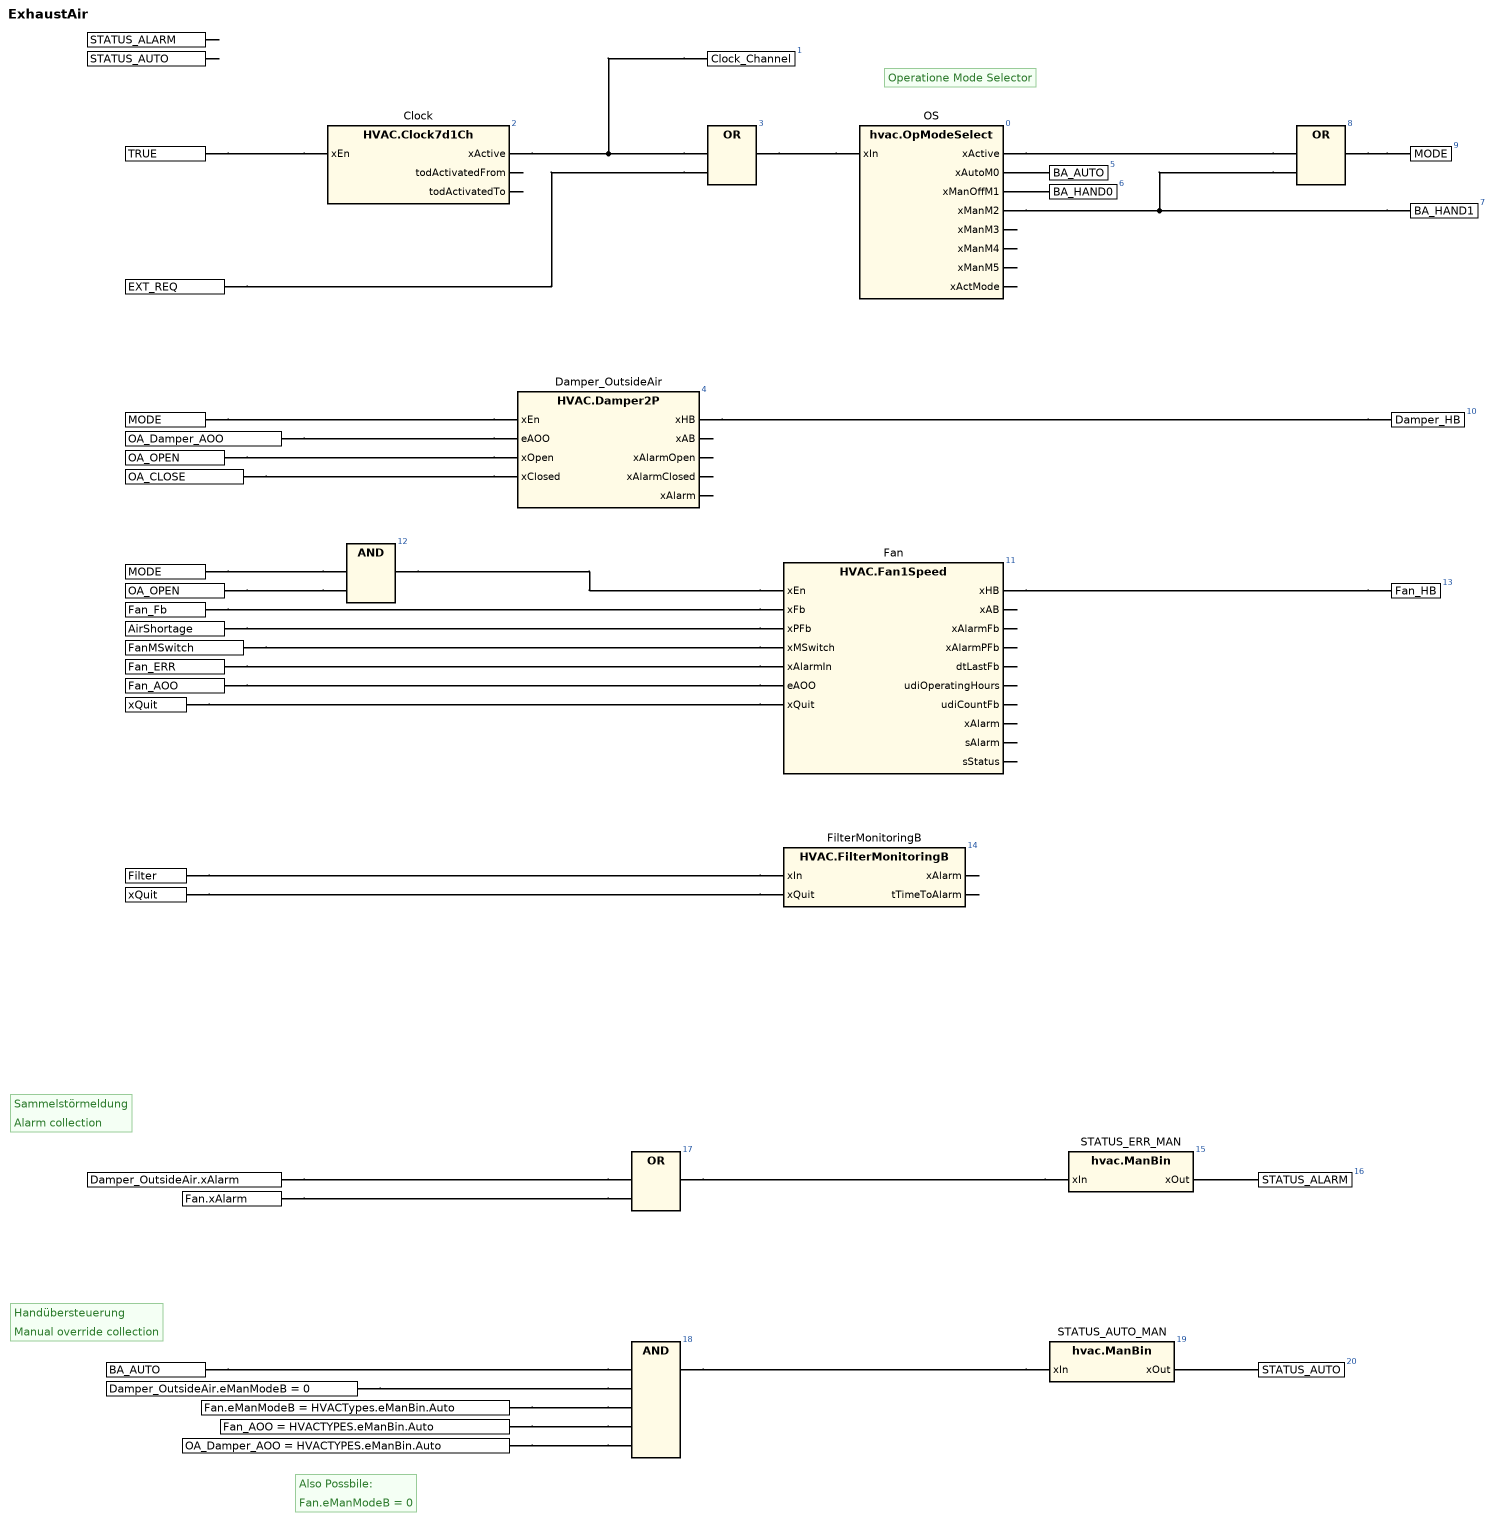
// note: 69 stored wires end on pins the file does not list and are not shown
// Operatione Mode Selector
// parameter OS.sTitleM2 := 'Manual On'
// parameter OS.sTitleM1 := 'Manual Off'
// parameter OS.sTitleM0 := 'Automatic'
// parameter OS.sTitle := 'Operation Mode'
// parameter OS.eMaxMode := HVAC.eOpMode.Mode2
OS(xIn := _w1); // hvac.OpModeSelect
Clock_Channel := Clock.xActive;
// parameter Clock.todSunTo := tod#00:00:00
// parameter Clock.todSunFrom := tod#00:00:00
// parameter Clock.todFriTo := tod#23:59:00
// parameter Clock.todFriFrom := tod#23:59:00
Clock(xEn := TRUE); // HVAC.Clock7d1Ch
_w1 := Clock.xActive OR EXT_REQ;
Damper_OutsideAir(xEn := MODE, eAOO := OA_Damper_AOO, xOpen := OA_OPEN, xClosed := OA_CLOSE); // HVAC.Damper2P
BA_AUTO := OS.xAutoM0;
BA_HAND0 := OS.xManOffM1;
BA_HAND1 := OS.xManM2;
MODE := OS.xActive OR OS.xManM2;
Damper_HB := Damper_OutsideAir.xHB;
Fan(
    xEn := _w2,
    xFb := Fan_Fb,
    xPFb := AirShortage,
    xMSwitch := FanMSwitch,
    xAlarmIn := Fan_ERR,
    eAOO := Fan_AOO,
    xQuit := xQuit); // HVAC.Fan1Speed
_w2 := MODE AND OA_OPEN;
Fan_HB := Fan.xHB;
FilterMonitoringB(xIn := Filter, xQuit := xQuit); // HVAC.FilterMonitoringB
STATUS_ERR_MAN(xIn := _w3); // hvac.ManBin
STATUS_ALARM := STATUS_ERR_MAN.xOut;
// Sammelstörmeldung
// Alarm collection
_w3 := Damper_OutsideAir.xAlarm OR Fan.xAlarm;
// Handübersteuerung
// Manual override collection
// Also Possbile:
// Fan.eManModeB = 0
STATUS_AUTO_MAN(xIn := BA_AUTO AND (Damper_OutsideAir.eManModeB = 0) AND (Fan.eManModeB = HVACTypes.eManBin.Auto) AND (Fan_AOO = HVACTYPES.eManBin.Auto) AND (OA_Damper_AOO = HVACTYPES.eManBin.Auto)); // hvac.ManBin
STATUS_AUTO := STATUS_AUTO_MAN.xOut;
// STATUS_ALARM: input not connected
// STATUS_AUTO: input not connected

END_FUNCTION_BLOCK

// Device/Application/AC_RMP/AC_PRG_RMP
//Code generated by Application Composer.
//Modifying generated code is not recommended!
PROGRAM AC_PRG_RMP
VAR
    itfRmpService2 : AC_PERSIST.AC.IRmpService2 := 0;
    xStartCyclicAction : BOOL;
    xIsActionOngoing : BOOL;
    xValid : BOOL;
    xValidEnd : BOOL := TRUE;
END_VAR

//Code generated by Application Composer.
//Modifying generated code is not recommended!
__QUERYINTERFACE(AC_RMP_Service, itfRmpService2);
IF itfRmpService2 <> 0 AND xValidEnd THEN
    xValid := itfRmpService2.GetIsActionOngoing(xIsActionOngoing=>xIsActionOngoing);
    IF NOT xValid OR (xValid AND xIsActionOngoing) THEN
        xStartCyclicAction := FALSE;
    ELSE
        xStartCyclicAction := itfRmpService2.SetIsActionOngoing(TRUE);
    END_IF
ELSE
    xStartCyclicAction := TRUE;
END_IF
IF xStartCyclicAction THEN
    AC_RMP_Service.CyclicCall() ;
END_IF
IF itfRmpService2 <> 0 AND (xStartCyclicAction OR NOT xValidEnd) THEN
    xValidEnd := itfRmpService2.SetIsActionOngoing(FALSE);
END_IF

END_PROGRAM

// Device/Application/AC_Std/AC_InitInternal
//Code generated by Application Composer.
//Modifying generated code is not recommended!
FUNCTION AC_InitInternal
VAR_INPUT
  bOnlineChange : BOOL ;
END_VAR
VAR
  hnd : AC_PERSIST.AC.ModuleHandle ;
END_VAR

//Code generated by Application Composer.
//Modifying generated code is not recommended!
AC_Environment.mtree := Module_Tree ;
AC_Environment.rmps := AC_RMP_Service ;
{IF defined(variable:AC_Environment.exts)}
	AC_Environment.exts := 0 ;
	AC_Environment.uiexts := 0 ;
{END_IF}
{IF defined(variable:AC_Environment.prsman)}
	AC_Environment.prsman := PersistenceManager;
{END_IF}
Module_Tree.Init(ADR(aNodes), 6);
hnd := Module_Tree.AddChild(0, PersistenceManager);
PersistenceManager.SetIdentification(ADR('PersistenceManager'), ADR(AC_PERSIST_PersistenceManager_INFO), 16#2610DE77, hnd, ADR(AC_Environment)) ;
hnd := Module_Tree.AddChild(PersistenceManager, PersistenceManager.INST_HVAC_Counter);
PersistenceManager.INST_HVAC_Counter.SetIdentification(ADR('HVAC_Counter'), ADR(AC_PERSIST_PersistenceChannel_INFO), 16#2610C9F2, hnd, ADR(AC_Environment)) ;
hnd := Module_Tree.AddChild(PersistenceManager, PersistenceManager.INST_HVAC_Parameter);
PersistenceManager.INST_HVAC_Parameter.SetIdentification(ADR('HVAC_Parameter'), ADR(AC_PERSIST_PersistenceChannel_INFO), 16#2610716B, hnd, ADR(AC_Environment)) ;
hnd := Module_Tree.AddChild(PersistenceManager.INST_HVAC_Counter, PersistenceManager.INST_HVAC_Counter.INST_ASCIIFileStorage);
PersistenceManager.INST_HVAC_Counter.INST_ASCIIFileStorage.SetIdentification(ADR('ASCIIFileStorage'), ADR(AC_PERSIST_ASCIIFileStorage_INFO), 16#2610E851, hnd, ADR(AC_Environment)) ;
hnd := Module_Tree.AddChild(PersistenceManager.INST_HVAC_Parameter, PersistenceManager.INST_HVAC_Parameter.INST_ASCIIFileStorage);
PersistenceManager.INST_HVAC_Parameter.INST_ASCIIFileStorage.SetIdentification(ADR('ASCIIFileStorage'), ADR(AC_PERSIST_ASCIIFileStorage_INFO), 16#261061FA, hnd, ADR(AC_Environment)) ;
PersistenceManager.uiNumberOfChannels := 2;
PersistenceManager.AC_ARRAY_pChannels[0] := PersistenceManager.INST_HVAC_Parameter;
PersistenceManager.AC_ARRAY_pChannels[1] := PersistenceManager.INST_HVAC_Counter;
PersistenceManager.pChannels := ADR(PersistenceManager.AC_ARRAY_pChannels);
PersistenceManager.INST_HVAC_Parameter.tPeriodicSaving := TIME#24h;
PersistenceManager.INST_HVAC_Parameter.xSaveOnChange := TRUE;
PersistenceManager.INST_HVAC_Parameter.xReadVarsDuringInit := TRUE;
PersistenceManager.INST_HVAC_Parameter.itfDataStorage := PersistenceManager.INST_HVAC_Parameter.INST_ASCIIFileStorage;
PersistenceManager.INST_HVAC_Counter.tPeriodicSaving := TIME#12h;
PersistenceManager.INST_HVAC_Counter.xSaveOnChange := FALSE;
PersistenceManager.INST_HVAC_Counter.xReadVarsDuringInit := TRUE;
PersistenceManager.INST_HVAC_Counter.itfDataStorage := PersistenceManager.INST_HVAC_Counter.INST_ASCIIFileStorage;
IF bOnlineChange THEN
    PersistenceManager.INST_HVAC_Parameter.xCompressTags := TRUE;
    PersistenceManager.INST_HVAC_Parameter.xConsistentCopyInHighPrioTask := FALSE;
    PersistenceManager.INST_HVAC_Parameter.xConvertVarsWithDifferentType := TRUE;
    PersistenceManager.INST_HVAC_Parameter.xIntegrityCheckBeforeReading := TRUE;
    PersistenceManager.INST_HVAC_Parameter.xSeparateArchivePerToplevelInstance := FALSE;
    PersistenceManager.INST_HVAC_Counter.xCompressTags := TRUE;
    PersistenceManager.INST_HVAC_Counter.xConsistentCopyInHighPrioTask := FALSE;
    PersistenceManager.INST_HVAC_Counter.xConvertVarsWithDifferentType := TRUE;
    PersistenceManager.INST_HVAC_Counter.xIntegrityCheckBeforeReading := TRUE;
    PersistenceManager.INST_HVAC_Counter.xSeparateArchivePerToplevelInstance := FALSE;
    PersistenceManager.INST_HVAC_Parameter.INST_ASCIIFileStorage.sArchive := '%CHANNEL_NAME%';
    PersistenceManager.INST_HVAC_Parameter.INST_ASCIIFileStorage.xDoubleStorage := FALSE;
    PersistenceManager.INST_HVAC_Parameter.INST_ASCIIFileStorage.udiMaximumFileSize := 0;
    PersistenceManager.INST_HVAC_Parameter.INST_ASCIIFileStorage.bySeparator := 9;
    PersistenceManager.INST_HVAC_Counter.INST_ASCIIFileStorage.sArchive := '%CHANNEL_NAME%';
    PersistenceManager.INST_HVAC_Counter.INST_ASCIIFileStorage.xDoubleStorage := FALSE;
    PersistenceManager.INST_HVAC_Counter.INST_ASCIIFileStorage.udiMaximumFileSize := 0;
    PersistenceManager.INST_HVAC_Counter.INST_ASCIIFileStorage.bySeparator := 9;
END_IF
PersistenceManager.Init(bOnlineChange);

END_FUNCTION

// Device/Application/AC_Std/AC_OnlineChange
//Code generated by Application Composer.
//Modifying generated code is not recommended!
{attribute 'linkalways'}
{attribute 'call_after_online_change_slot' := '1234'}
FUNCTION AC_OnlineChange

//Code generated by Application Composer.
//Modifying generated code is not recommended!
PersistenceManager.OnBeforeOnlineChange();
AC_InitInternal(TRUE);
PersistenceManager.OnAfterOnlineChange();

END_FUNCTION

// Device/Application/AC_FBs/AC_PersistenceManager_HVAC_Parameter
//Code generated by Application Composer.
//Modifying generated code is not recommended!
FUNCTION_BLOCK AC_PersistenceManager_HVAC_Parameter EXTENDS AC_PERSIST.PersistenceChannel
VAR_INPUT 
    INST_ASCIIFileStorage : AC_PERSIST.ASCIIFileStorage;
END_VAR

//Code generated by Application Composer.
//Modifying generated code is not recommended!
SUPER^();

END_FUNCTION_BLOCK

// Device/Application/AC_FBs/AC_PersistenceManager_HVAC_Counter
//Code generated by Application Composer.
//Modifying generated code is not recommended!
FUNCTION_BLOCK AC_PersistenceManager_HVAC_Counter EXTENDS AC_PERSIST.PersistenceChannel
VAR_INPUT 
    INST_ASCIIFileStorage : AC_PERSIST.ASCIIFileStorage;
END_VAR

//Code generated by Application Composer.
//Modifying generated code is not recommended!
SUPER^();

END_FUNCTION_BLOCK

// Device/Application/AC_FBs/AC_PersistenceManager
//Code generated by Application Composer.
//Modifying generated code is not recommended!
FUNCTION_BLOCK AC_PersistenceManager EXTENDS AC_PERSIST.PersistenceManager
VAR_INPUT 
    INST_HVAC_Parameter : AC_PersistenceManager_HVAC_Parameter;
    INST_HVAC_Counter : AC_PersistenceManager_HVAC_Counter;
    AC_ARRAY_pChannels : ARRAY[0..1] OF AC_PERSIST.IPersistenceChannel;
END_VAR

//Code generated by Application Composer.
//Modifying generated code is not recommended!
SUPER^();

END_FUNCTION_BLOCK

// Device/Application/AC_Std/AC_Init
//Code generated by Application Composer.
//Modifying generated code is not recommended!
{attribute 'linkalways'}
{attribute 'call_after_global_init_slot' := '1234'}
FUNCTION AC_Init

//Code generated by Application Composer.
//Modifying generated code is not recommended!
AC_InitInternal(FALSE);

END_FUNCTION

// Device/Application/Visu/3_Settings/Settings_Start
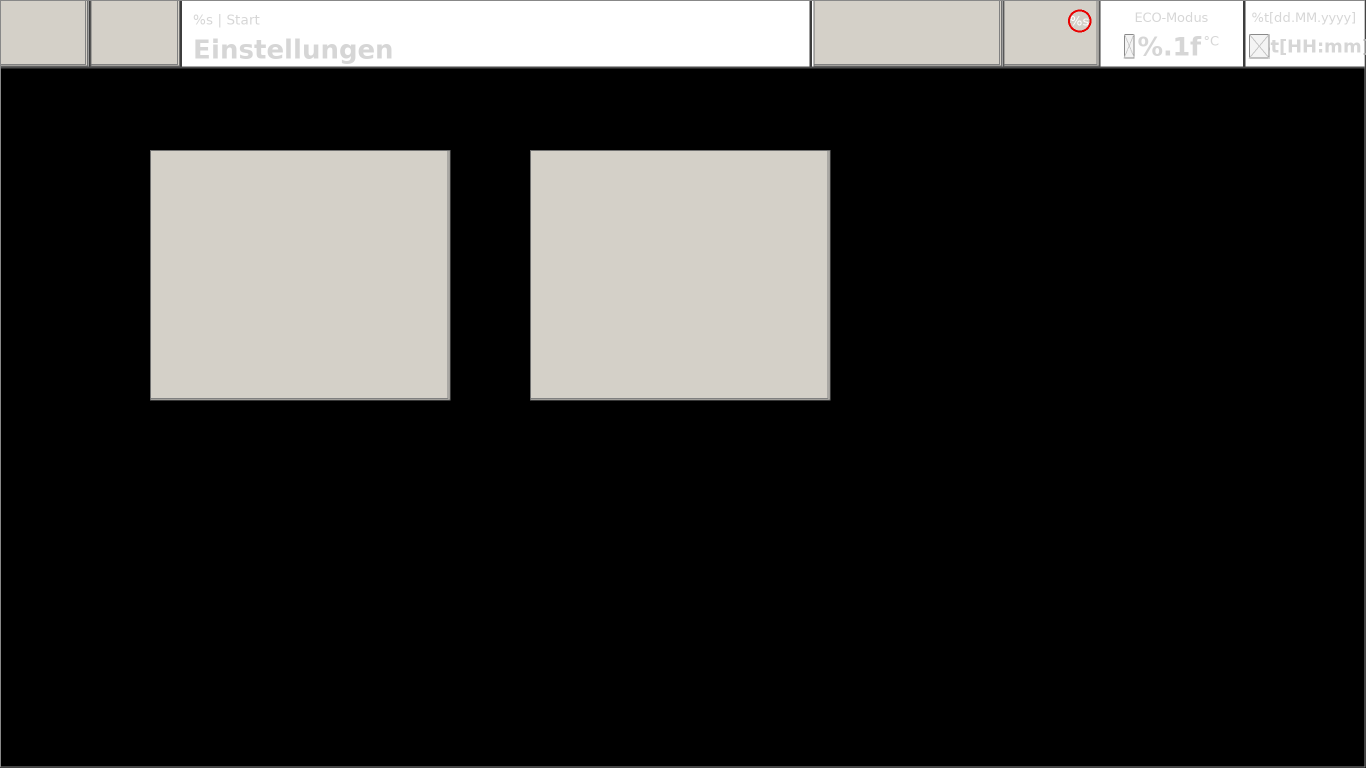
VISUALIZATION Settings_Start  // 1366x768
    Frame (0,0 1366x70)
        shows Header_Frame()
    Rectangle (190,5 545x30), "%s | Start", text variable: PRG.GebVar
    Rectangle (190,32 545x35), "Einstellungen"
    Rectangle (150,150 300x250)
    Rectangle (150,175 300x30), "PERSISTENCE"
    Image (235,230 126x125), image: HVACV.HVACImage.book
    Button (150,150 300x250)
        OnMouseClick:  Assign=Settings_Persistence, Type=Assignment
    Rectangle (530,150 300x250)
    Rectangle (530,175 300x30), "MAN INFO"
    Image (635,230 96x96), image: HVACV.HVACImage.edit2
    RoundedRectangle (620,350 120x30), "inaktiv", invisible if: Main.ManInfo.xManActive
    RoundedRectangle (620,350 120x30), "aktiv", invisible if: NOT Main.ManInfo.xManActive
    Button (530,150 300x250)
        OnMouseClick:  Assign=Settings_MANInfo, Type=Assignment
END_VISUALIZATION

// Device/Application/Visu/0_Alarm/Alarm_Start
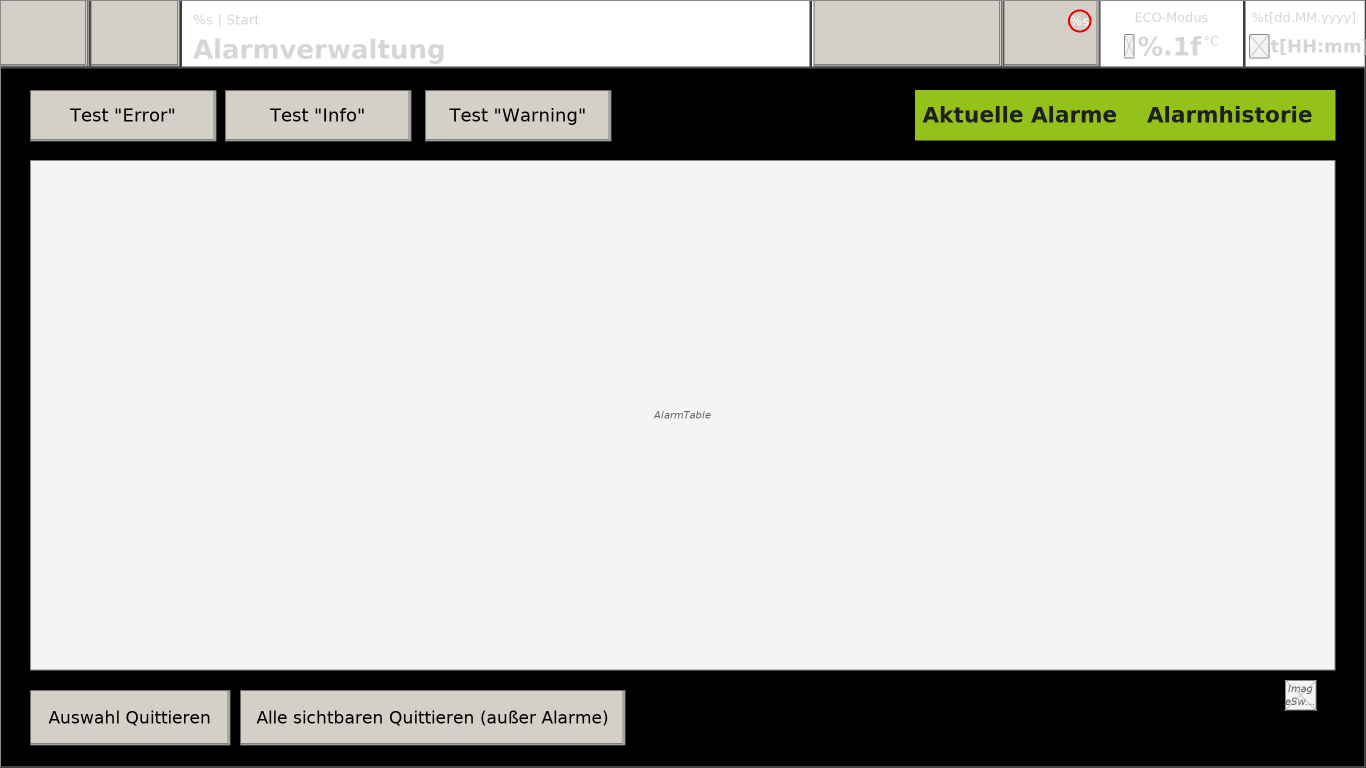
VISUALIZATION Alarm_Start  // 1366x768
VAR_IN_OUT
	
END_VAR

VAR
	bAckSel : BOOL;
	bAckVisible : BOOL;
	bHistory : BOOL;
	bFreezeScrlPos : BOOL;
	iColSort : INT :=2;
	xColSort : BOOL :=FALSE;
END_VAR
    Frame (0,0 1366x70)
        shows Header_Frame()
    Rectangle (190,5 545x30), "%s | Start", text variable: PRG.GebVar
    Rectangle (190,32 545x35), "Alarmverwaltung"
    AlarmTable (30,160 1305x510)
        Column[0]: ColumnTitle=Symbol
        Column[1]: ColumnTitle=Meldungstext
        Column[2]: ColumnTitle=Gekommen
        Column[3]: ColumnTitle=Gegangen
        Column[4]: ColumnTitle=Typ
        Column[5]: ColumnTitle=Status
        p1521930926: __All
        p1663851261: __All
        p428520879: bAckSel
        p2607059081: bAckVisible
        p3266827225: bHistory
        p3894972949: bFreezeScrlPos
        p4280204719: iColSort
        p3852279139: xColSort
    Button (30,690 200x55), "Auswahl Quittieren", invisible if: bHistory
        toggle bAckSel
    Button (240,690 385x55), "Alle sichtbaren Quittieren (außer Alarme)", invisible if: bHistory
        toggle bAckVisible
    ImageSwitcher (1285,680 31x30), variable: bFreezeScrlPos, background image: HVACV.HVACImage.lock, image: HVACV.HVACImage.lockopen, behaviour: TOGGLE
    Rectangle (915,90 210x50), "Aktuelle Alarme"
        OnMouseClick: execute { bHistory := FALSE; }
    Rectangle (915,90 210x50), "Aktuelle Alarme", invisible if: bHistory
        OnMouseClick: execute { bHistory := FALSE; }
    Rectangle (1125,90 210x50), "Alarmhistorie"
        OnMouseClick: execute { bHistory := TRUE; }
    Rectangle (1125,90 210x50), "Alarmhistorie", invisible if: NOT(bHistory)
        OnMouseClick: execute { bHistory := TRUE; }
    Button (30,90 186x51), "Test "Error"", colour toggle: Main.xErrorTest
        OnMouseClick:  ToggleVariable=Main.xErrorTest
    Button (225,90 186x51), "Test "Info"", colour toggle: Main.xInfoTest
        OnMouseClick:  ToggleVariable=Main.xInfoTest
    Button (425,90 186x51), "Test "Warning"", colour toggle: Main.xWarningTest
        OnMouseClick:  ToggleVariable=Main.xWarningTest
END_VISUALIZATION

// Device/Application/Macros and frames/HeatingCircuit/HeatCurve4P_DN
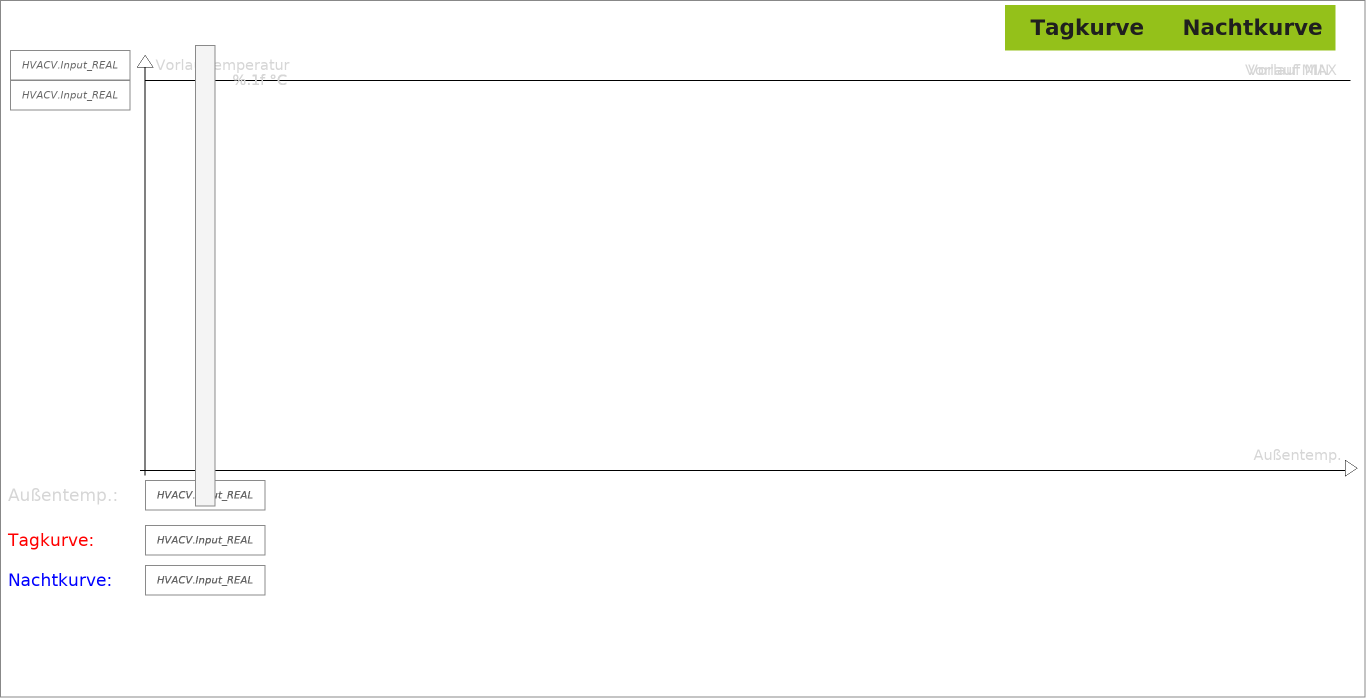
VISUALIZATION HeatCurve4P_DN  // 1366x698
VAR_IN_OUT
	FB_HeatCurve4P_DN : HVAC.HeatCurve4P_DN;
END_VAR

VAR
	Umschaltung_Tag_Nacht : BOOL := TRUE; // DAY  =TRUE NIGHT=FALSE
END_VAR
    Line (205,90) (205,465)
        p3560616238: FB_HeatCurve4P_DN._iVisu_To2
    Line (205,90) (205,465)
        p3560616238: FB_HeatCurve4P_DN._iVisu_To1
    Line (205,90) (205,465)
        p3560616238: FB_HeatCurve4P_DN._iVisu_To3
    Line (205,90) (205,465)
        p3560616238: FB_HeatCurve4P_DN._iVisu_To4
    Line (140,470) (1350,470)
    Line (145,475) (145,65)
    Line (145,80) (1350,80)
        p2738717112: FB_HeatCurve4P_DN._iVisu_VL_MAX
    Line (145,80) (1350,80)
        p2738717112: FB_HeatCurve4P_DN._iVisu_VL_Min
    Polygon (137,67) (153,67) (145,55)
    Polygon (1345,460) (1345,476) (1357,468)
    Line (205,80) (305,80)
        p874137650: FB_HeatCurve4P_DN._iVisu_To2 - 100
        p1126004900: FB_HeatCurve4P_DN._iVisu_W2_TAG
        p3528305787: FB_HeatCurve4P_DN._iVisu_To1
        p2773130477: FB_HeatCurve4P_DN._iVisu_W1_TAG
    Frame (145,525 120x30)
        shows HVACV.Input_REAL(rValue := FB_HeatCurve4P_DN.rW1Day, bDecimals := 1, sUnit := '°C', rMinInputVisu := 0, rMaxInputVisu := 100)
        p3560616238: FB_HeatCurve4P_DN._iVisu_To1
    Frame (145,565 120x30)
        shows HVACV.Input_REAL(rValue := FB_HeatCurve4P_DN.rW1Night, bDecimals := 1, sUnit := '°C', rMinInputVisu := 0, rMaxInputVisu := 100)
        p3560616238: FB_HeatCurve4P_DN._iVisu_To1
    Frame (145,480 120x30)
        shows HVACV.Input_REAL(rValue := FB_HeatCurve4P_DN.rTo1, bDecimals := 1, sUnit := '°C', rMinInputVisu := -50, rMaxInputVisu := FB_HeatCurve4P_DN.rTo2 -2)
        p3560616238: FB_HeatCurve4P_DN._iVisu_To1
    Rectangle (5,525 135x30), "Tagkurve:"
    Rectangle (5,565 135x30), "Nachtkurve:"
    Rectangle (5,480 135x30), "Außentemp.:"
    Frame (145,525 120x30)
        shows HVACV.Input_REAL(rValue := FB_HeatCurve4P_DN.rW2Day, bDecimals := 1, sUnit := '°C', rMinInputVisu := 0, rMaxInputVisu := 100)
        p3560616238: FB_HeatCurve4P_DN._iVisu_To2
    Frame (145,525 120x30)
        shows HVACV.Input_REAL(rValue := FB_HeatCurve4P_DN.rW3Day, bDecimals := 1, sUnit := '°C', rMinInputVisu := 0, rMaxInputVisu := 100)
        p3560616238: FB_HeatCurve4P_DN._iVisu_To3
    Frame (145,525 120x30)
        shows HVACV.Input_REAL(rValue := FB_HeatCurve4P_DN.rW4Day, bDecimals := 1, sUnit := '°C', rMinInputVisu := 0, rMaxInputVisu := 100)
        p3560616238: FB_HeatCurve4P_DN._iVisu_To4
    Frame (145,565 120x30)
        shows HVACV.Input_REAL(rValue := FB_HeatCurve4P_DN.rW2Night, bDecimals := 1, sUnit := '°C', rMinInputVisu := 0, rMaxInputVisu := 100)
        p3560616238: FB_HeatCurve4P_DN._iVisu_To2
    Frame (145,565 120x30)
        shows HVACV.Input_REAL(rValue := FB_HeatCurve4P_DN.rW3Night, bDecimals := 1, sUnit := '°C', rMinInputVisu := 0, rMaxInputVisu := 100)
        p3560616238: FB_HeatCurve4P_DN._iVisu_To3
    Frame (145,565 120x30)
        shows HVACV.Input_REAL(rValue := FB_HeatCurve4P_DN.rW4Night, bDecimals := 1, sUnit := '°C', rMinInputVisu := 0, rMaxInputVisu := 100)
        p3560616238: FB_HeatCurve4P_DN._iVisu_To4
    Frame (145,480 120x30)
        shows HVACV.Input_REAL(rValue := FB_HeatCurve4P_DN.rTo2, bDecimals := 1, sUnit := '°C', rMinInputVisu := FB_HeatCurve4P_DN.rTo1 +2, rMaxInputVisu := FB_HeatCurve4P_DN.rTo3 -2)
        p3560616238: FB_HeatCurve4P_DN._iVisu_To2
    Frame (145,480 120x30)
        shows HVACV.Input_REAL(rValue := FB_HeatCurve4P_DN.rTo3, bDecimals := 1, sUnit := '°C', rMinInputVisu := FB_HeatCurve4P_DN.rTo2 +2, rMaxInputVisu := FB_HeatCurve4P_DN.rTo4 -2)
        p3560616238: FB_HeatCurve4P_DN._iVisu_To3
    Frame (145,480 120x30)
        shows HVACV.Input_REAL(rValue := FB_HeatCurve4P_DN.rTo4, bDecimals := 1, sUnit := '°C', rMinInputVisu := FB_HeatCurve4P_DN.rTo3 + 2, rMaxInputVisu := 50)
        p3560616238: FB_HeatCurve4P_DN._iVisu_To4
    Rectangle (1245,440 105x30), "Außentemp."
    Rectangle (145,50 155x30), "Vorlauftemperatur"
    Frame (10,80 120x30)
        shows HVACV.Input_REAL(rValue := FB_HeatCurve4P_DN.rSupplyTempMin, bDecimals := 1, sUnit := '°C', rMinInputVisu := 0, rMaxInputVisu := FB_HeatCurve4P_DN.rSupplyTempMax)
        p2738717112: FB_HeatCurve4P_DN._iVisu_VL_Min
    Frame (10,50 120x30)
        shows HVACV.Input_REAL(rValue := FB_HeatCurve4P_DN.rSupplyTempMax, bDecimals := 1, sUnit := '°C', rMinInputVisu := FB_HeatCurve4P_DN.rSupplyTempMin, rMaxInputVisu := 100)
        p2738717112: FB_HeatCurve4P_DN._iVisu_VL_MAX
    Line (205,80) (305,80)
        p874137650: FB_HeatCurve4P_DN._iVisu_To3 - 100
        p1126004900: FB_HeatCurve4P_DN._iVisu_W3_TAG
        p3528305787: FB_HeatCurve4P_DN._iVisu_To2
        p2773130477: FB_HeatCurve4P_DN._iVisu_W2_TAG
    Line (205,80) (305,80)
        p874137650: FB_HeatCurve4P_DN._iVisu_To4 - 100
        p1126004900: FB_HeatCurve4P_DN._iVisu_W4_TAG
        p3528305787: FB_HeatCurve4P_DN._iVisu_To3
        p2773130477: FB_HeatCurve4P_DN._iVisu_W3_TAG
    Rectangle (1240,55 105x30), "Vorlauf MAX"
        p2738717112: FB_HeatCurve4P_DN._iVisu_VL_MAX
    Rectangle (1235,55 105x30), "Vorlauf MIN"
        p2738717112: FB_HeatCurve4P_DN._iVisu_VL_Min
    Line (205,80) (305,80)
        p874137650: FB_HeatCurve4P_DN._iVisu_To2 - 100
        p1126004900: FB_HeatCurve4P_DN._iVisu_W2_NACHT
        p3528305787: FB_HeatCurve4P_DN._iVisu_To1
        p2773130477: FB_HeatCurve4P_DN._iVisu_W1_NACHT
    Line (205,80) (305,80)
        p874137650: FB_HeatCurve4P_DN._iVisu_To3 - 100
        p1126004900: FB_HeatCurve4P_DN._iVisu_W3_NACHT
        p3528305787: FB_HeatCurve4P_DN._iVisu_To2
        p2773130477: FB_HeatCurve4P_DN._iVisu_W2_NACHT
    Line (205,80) (305,80)
        p874137650: FB_HeatCurve4P_DN._iVisu_To4 - 100
        p1126004900: FB_HeatCurve4P_DN._iVisu_W4_NACHT
        p3528305787: FB_HeatCurve4P_DN._iVisu_To3
        p2773130477: FB_HeatCurve4P_DN._iVisu_W3_NACHT
    Group (195,45 100x461), invisible if: (FB_HeatCurve4P_DN.rSupplyTempMaxScale <> 90) OR (Umschaltung_Tag_Nacht)
        p3560616238: FB_HeatCurve4P_DN._iVisu_To1
        Slider (0,0 20x461), variable: FB_HeatCurve4P_DN.rW1Night, scale 0..90
        Rectangle (30,20 70x30), "%.1f °C", text variable: FB_HeatCurve4P_DN.rW1Night
            p2738717112: FB_HeatCurve4P_DN._iVisu_W1_NACHT
    Group (195,45 100x461), invisible if: (FB_HeatCurve4P_DN.rSupplyTempMaxScale <> 90) OR (Umschaltung_Tag_Nacht)
        p3560616238: FB_HeatCurve4P_DN._iVisu_To2
        Slider (0,0 20x461), variable: FB_HeatCurve4P_DN.rW2Night, scale 0..90
        Rectangle (30,20 70x30), "%.1f °C", text variable: FB_HeatCurve4P_DN.rW2Night
            p2738717112: FB_HeatCurve4P_DN._iVisu_W2_NACHT
    Group (195,45 100x461), invisible if: (FB_HeatCurve4P_DN.rSupplyTempMaxScale <> 90) OR (Umschaltung_Tag_Nacht)
        p3560616238: FB_HeatCurve4P_DN._iVisu_To3
        Slider (0,0 20x461), variable: FB_HeatCurve4P_DN.rW3Night, scale 0..90
        Rectangle (30,20 70x30), "%.1f °C", text variable: FB_HeatCurve4P_DN.rW3Night
            p2738717112: FB_HeatCurve4P_DN._iVisu_W3_NACHT
    Group (195,45 100x461), invisible if: (FB_HeatCurve4P_DN.rSupplyTempMaxScale <> 90) OR (Umschaltung_Tag_Nacht)
        p3560616238: FB_HeatCurve4P_DN._iVisu_To4
        Slider (0,0 20x461), variable: FB_HeatCurve4P_DN.rW4Night, scale 0..90
        Rectangle (30,20 70x30), "%.1f °C", text variable: FB_HeatCurve4P_DN.rW4Night
            p2738717112: FB_HeatCurve4P_DN._iVisu_W4_NACHT
    Group (195,45 100x461), invisible if: (FB_HeatCurve4P_DN.rSupplyTempMaxScale <> 90) OR (NOT Umschaltung_Tag_Nacht)
        p3560616238: FB_HeatCurve4P_DN._iVisu_To1
        Slider (0,0 20x461), variable: FB_HeatCurve4P_DN.rW1Day, scale 0..90
        Rectangle (30,20 70x30), "%.1f °C", text variable: FB_HeatCurve4P_DN.rW1Day
            p2738717112: FB_HeatCurve4P_DN._iVisu_W1_TAG
    Group (195,45 100x461), invisible if: (FB_HeatCurve4P_DN.rSupplyTempMaxScale <> 90) OR (NOT Umschaltung_Tag_Nacht)
        p3560616238: FB_HeatCurve4P_DN._iVisu_To2
        Slider (0,0 20x461), variable: FB_HeatCurve4P_DN.rW2Day, scale 0..90
        Rectangle (30,20 70x30), "%.1f °C", text variable: FB_HeatCurve4P_DN.rW2Day
            p2738717112: FB_HeatCurve4P_DN._iVisu_W2_TAG
    Group (195,45 100x461), invisible if: (FB_HeatCurve4P_DN.rSupplyTempMaxScale <> 90) OR (NOT Umschaltung_Tag_Nacht)
        p3560616238: FB_HeatCurve4P_DN._iVisu_To3
        Slider (0,0 20x461), variable: FB_HeatCurve4P_DN.rW3Day, scale 0..90
        Rectangle (30,20 70x30), "%.1f °C", text variable: FB_HeatCurve4P_DN.rW3Day
            p2738717112: FB_HeatCurve4P_DN._iVisu_W3_TAG
    Group (195,45 100x461), invisible if: (FB_HeatCurve4P_DN.rSupplyTempMaxScale <> 90) OR (NOT Umschaltung_Tag_Nacht)
        p3560616238: FB_HeatCurve4P_DN._iVisu_To4
        Slider (0,0 20x461), variable: FB_HeatCurve4P_DN.rW4Day, scale 0..90
        Rectangle (30,20 70x30), "%.1f °C", text variable: FB_HeatCurve4P_DN.rW4Day
            p2738717112: FB_HeatCurve4P_DN._iVisu_W4_TAG
    Rectangle (1005,5 165x45), "Tagkurve", invisible if: FB_HeatCurve4P_DN.rSupplyTempMaxScale <> 90
        OnMouseClick:  ToggleVariable=Umschaltung_Tag_Nacht
    Rectangle (1005,5 165x45), "Tagkurve", invisible if: (NOT Umschaltung_Tag_Nacht) OR (FB_HeatCurve4P_DN.rSupplyTempMaxScale <> 90)
        OnMouseClick:  ToggleVariable=Umschaltung_Tag_Nacht
    Rectangle (1170,5 165x45), "Nachtkurve", invisible if: FB_HeatCurve4P_DN.rSupplyTempMaxScale <> 90
        OnMouseClick:  ToggleVariable=Umschaltung_Tag_Nacht
    Rectangle (1170,5 165x45), "Nachtkurve", invisible if: (Umschaltung_Tag_Nacht) Or (FB_HeatCurve4P_DN.rSupplyTempMaxScale <> 90)
        OnMouseClick:  ToggleVariable=Umschaltung_Tag_Nacht
END_VISUALIZATION

// Device/Application/Visu/Header_Frame
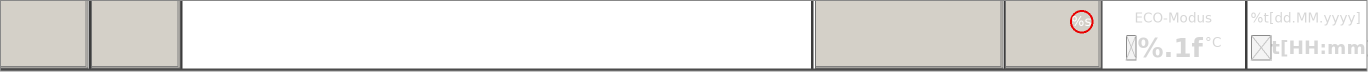
VISUALIZATION Header_Frame  // 1368x72
    Rectangle (0,66 1366x4)
    Rectangle (0,0 1366x68)
    Rectangle (1246,8 120x20), "%t[dd.MM.yyyy]"
    Rectangle (1266,35 95x25), "%t[HH:mm]"
    Rectangle (1245,0 2x68)
    Rectangle (89,0 2x68)
    Rectangle (1100,0 2x68)
    Rectangle (1101,8 145x20), "ECO-Modus"
    Rectangle (1136,35 70x26), "%.1f", text variable: Main.OutsideTemp_TS
    Image (1126,35 10x25), image: HVACV.HVACImage.thermometer1
    Rectangle (1201,35 25x15), "°C"
    Image (110,9 52x52), image: HVACV.HVACImage.back
    Image (20,9 52x52), image: HVACV.HVACImage.home
    Rectangle (180,0 2x68)
    Button (0,0 88x68)
        OnMouseClick:  Assign=Start, Type=Assignment
    Button (91,0 89x68)
        OnMouseClick:  Type=Previous
        OnMouseClick: FrameSelectionChange Selection=Selection=-1, GlobSel=IndExpr=0, AssignDir=Objekte.GenElemInst_23, AssignType=Directly, SelType=Globally
    Rectangle (1004,0 2x68)
    Rectangle (811,0 2x68)
    RoundedRectangle (826,30 140x30), "%s", text variable: VisuElems.CurrentFullUserName
    RoundedRectangle (961,30 30x30)
    Polygon (956,45) (962,51) (962,40)
    Line (956,45) (961,40)
    Line (956,45) (961,50)
    Image (966,35 19x21), image: HVACV.HVACImage.user_dark
    Rectangle (811,6 195x20), "angemeldet als"
    Button (815,0 188x68)
        OnMouseClick:  Type=Login
    Image (1251,35 20x25), image: HVACV.HVACImage.clock
    Image (1030,15 51x51), image: HVACV.HVACImage.warning
    Ellipse (1070,10 23x23), "%s", text variable: Main.AlarmCounter_Warning.iActive, invisible if: (Main.AlarmCounter.iActive > 0) OR (Main.AlarmCounter_Warning.iActive = 0)
    Image (1030,15 51x51), invisible if: (Main.AlarmCounter.iActive > 0) OR (Main.AlarmCounter_Warning.iActive = 0), image: HVACV.HVACImage.warning_orange
    Image (1030,15 51x51), invisible if: NOT Main.xAlarme_blinker, image: HVACV.HVACImage.warning_red
    Button (1005,0 96x68)
        OnMouseClick:  Assign=Alarm_Start, Type=Assignment
    Ellipse (1070,10 23x23), "%s", text variable: Main.AlarmCounter.iActive, invisible if: NOT(Main.AlarmCounter.iActive > 0)
    hotkey  Id=481037385728, Key=KeyDown=True, KeyName=ESCAPE, VisuElemId=1
    hotkey  Id=481038434304, Key=KeyName=ESCAPE, VisuElemId=1
    hotkey  Id=481039482880, Key=KeyDown=True, KeyName=BACKSPACE, VisuElemId=38
    hotkey  Id=481040531456, Key=KeyName=BACKSPACE, VisuElemId=38
END_VISUALIZATION

// Device/Application/Start
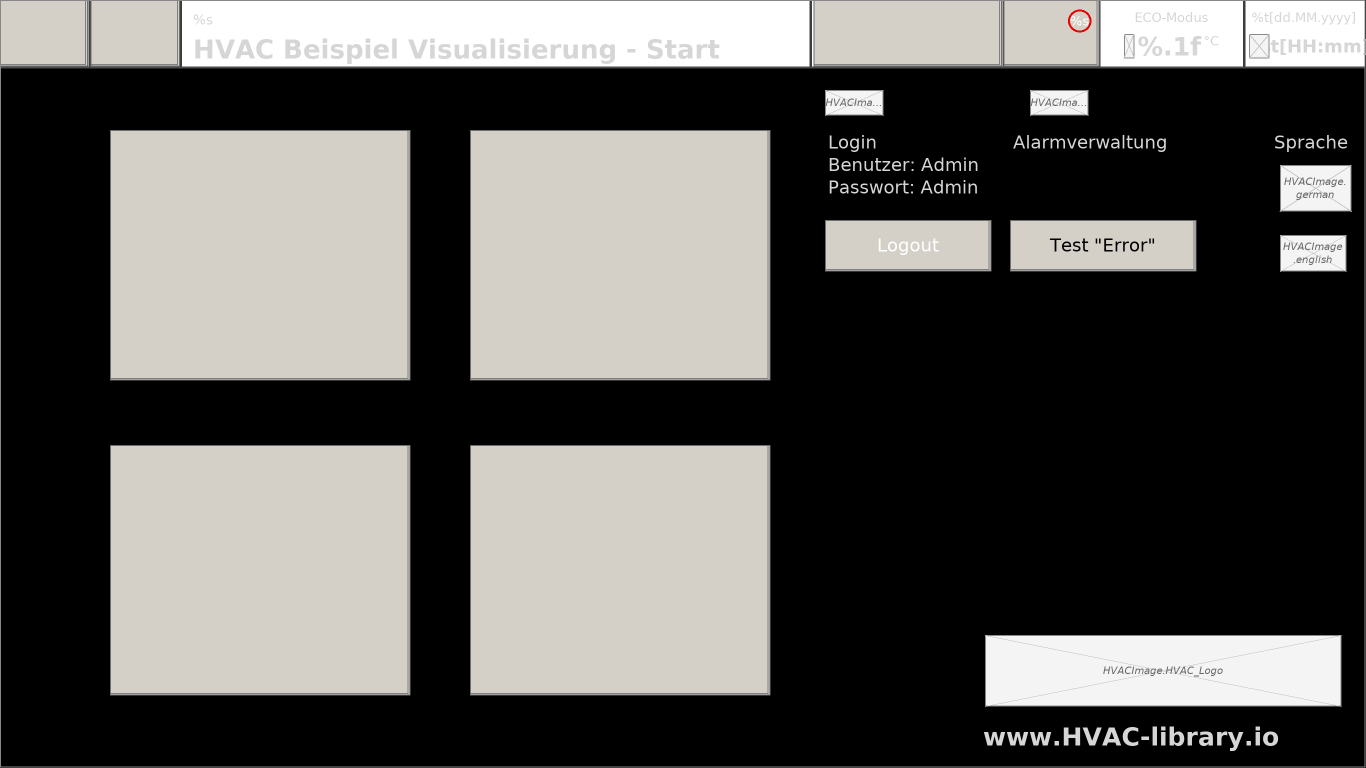
VISUALIZATION Start  // 1366x768
    Rectangle (110,130 300x250)
    Rectangle (110,150 300x30), "OBJEKTE"
    Image (210,195 98x111), image: HVACV.HVACImage.object
    RoundedRectangle (220,335 79x30), "Störung", invisible if: NOT(Main.AlarmCounter.iActive > 0)
    RoundedRectangle (225,335 71x30), "hand", invisible if: (Main.AlarmCounter.iActive > 0) OR (Main.AlarmCounter_Warning.iActive = 0)
    RoundedRectangle (205,335 114x30), "Automatik", invisible if: (Main.AlarmCounter.iActive > 0) OR (Main.AlarmCounter_Warning.iActive > 0)
    Button (110,130 300x250)
        OnMouseClick:  Assign=Objects_Start, Type=Assignment
    Frame (0,0 1366x70)
        shows Header_Frame()
    Button (1010,220 186x51), "Test "Error"", colour toggle: Main.xErrorTest
        OnMouseClick:  ToggleVariable=Main.xErrorTest
    Rectangle (110,445 300x250)
    Rectangle (110,465 300x30), "EINSTELLUNGEN"
    Image (185,525 136x106), image: HVACV.HVACImage.settings
    Button (110,445 300x250)
        OnMouseClick:  Assign=Settings_Start, Type=Assignment
    Rectangle (190,5 545x30), "%s", text variable: PRG.GebVar
    Rectangle (190,32 545x35), "HVAC Beispiel Visualisierung - Start"
    Image (985,635 356x71), image: HVACImage.HVAC_Logo
        OnMouseClick:  ExecuteCommand=ExecuteCommand=[Command=NavigateURL, Value='https://hvac-library.io/de/']
    Image (1280,235 66x36), image: HVACImage.english
        OnMouseClick:  ChangeLanguage=EN
    Image (1280,165 71x46), image: HVACImage.german
        OnMouseClick:  ChangeLanguage=DE
    Rectangle (825,130 236x91), "Login Benutzer: Admin Passwort: Admin"
    Button (825,220 166x51), "Logout"
        OnMouseClick:  Type=Logout
    Rectangle (1010,130 236x91), "Alarmverwaltung"
    Rectangle (1230,130 121x41), "Sprache"
    Image (825,90 58x25), angle 90, image: HVACImage.arrow_left
    Image (1030,90 58x25), angle 90, image: HVACImage.arrow_left
    Rectangle (470,130 300x250)
    Rectangle (470,150 300x30), "ZEITPROGRAMME"
    Image (570,210 101x111), image: HVACV.HVACImage.clock2
    Button (470,130 300x250)
        OnMouseClick:  Assign=Clock_Settings_Start, Type=Assignment
    Rectangle (470,445 300x250)
    Rectangle (470,465 300x30), "AUßENKONDITIONEN"
    Image (565,525 106x116), image: HVACV.HVACImage.weather
    Button (470,445 300x250)
        OnMouseClick:  Assign=Weather_Start, Type=Assignment
    Rectangle (980,720 351x46), "www.HVAC-library.io"
        OnMouseClick:  ExecuteCommand=ExecuteCommand=[Command=NavigateURL, Value='https://hvac-library.io/de/']
END_VISUALIZATION

// Device/Application/Visu/1_Objects/Room_1/Clock_Room_1
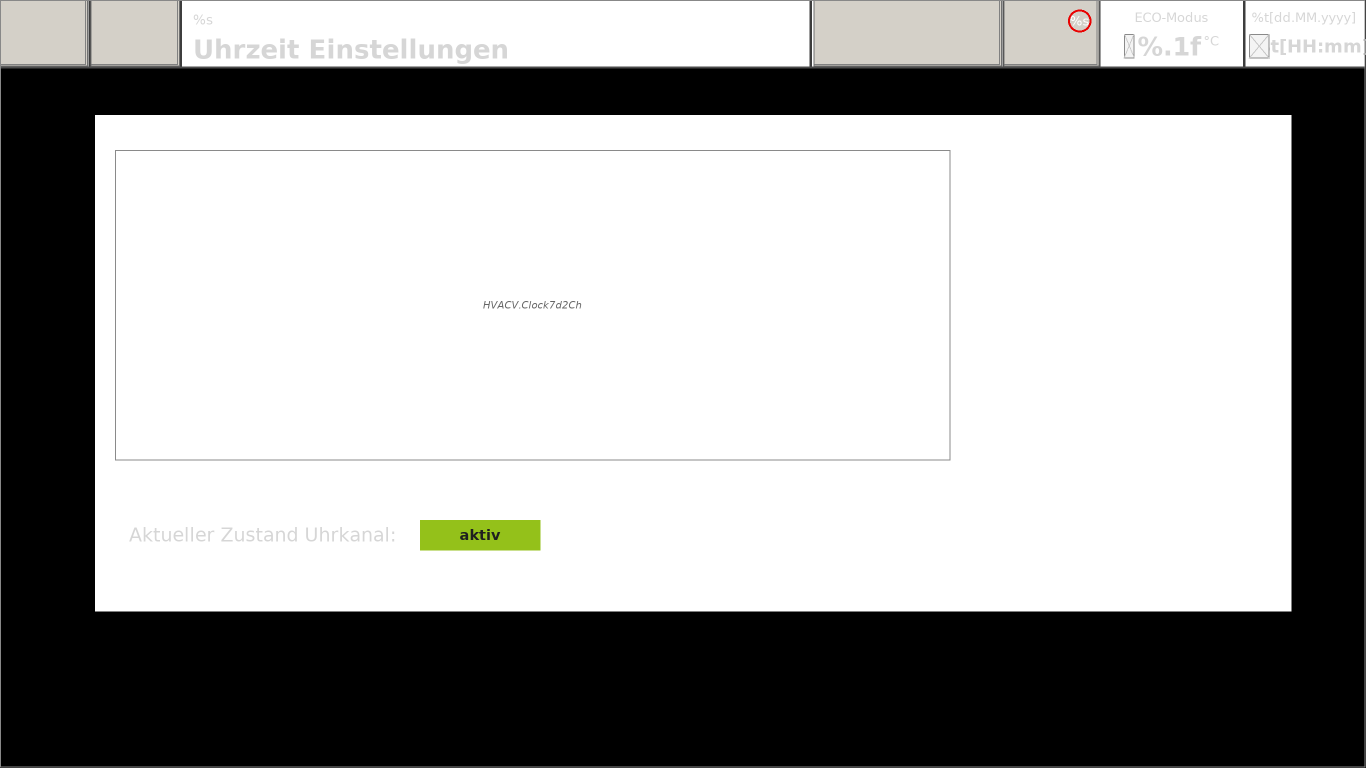
VISUALIZATION Clock_Room_1  // 1366x768
    Rectangle (95,115 1196x496)
    Frame (0,0 1366x70)
        shows Header_Frame()
    Rectangle (190,5 545x30), "%s", text variable: CONCAT( CONCAT(PRG.GebVar, ' | Start | Objekte | '), Prg.Room_1.Titel)
    Rectangle (190,32 545x35), "Uhrzeit Einstellungen"
    RoundedRectangle (420,520 120x30), "inaktiv", invisible if: PRG.Room_1.Clock.xActive
    RoundedRectangle (420,520 120x30), "aktiv", invisible if: NOT PRG.Room_1.Clock.xActive
    Rectangle (115,520 296x30), "Aktueller Zustand Uhrkanal:"
    Frame (115,150 835x310)
        shows HVACV.Clock7d2Ch(FB_Clock7d2Ch := PRG.Room_1.Clock)
END_VISUALIZATION

// Device/Application/Macros and frames/Room_DE/Zone_F_Therm_Start
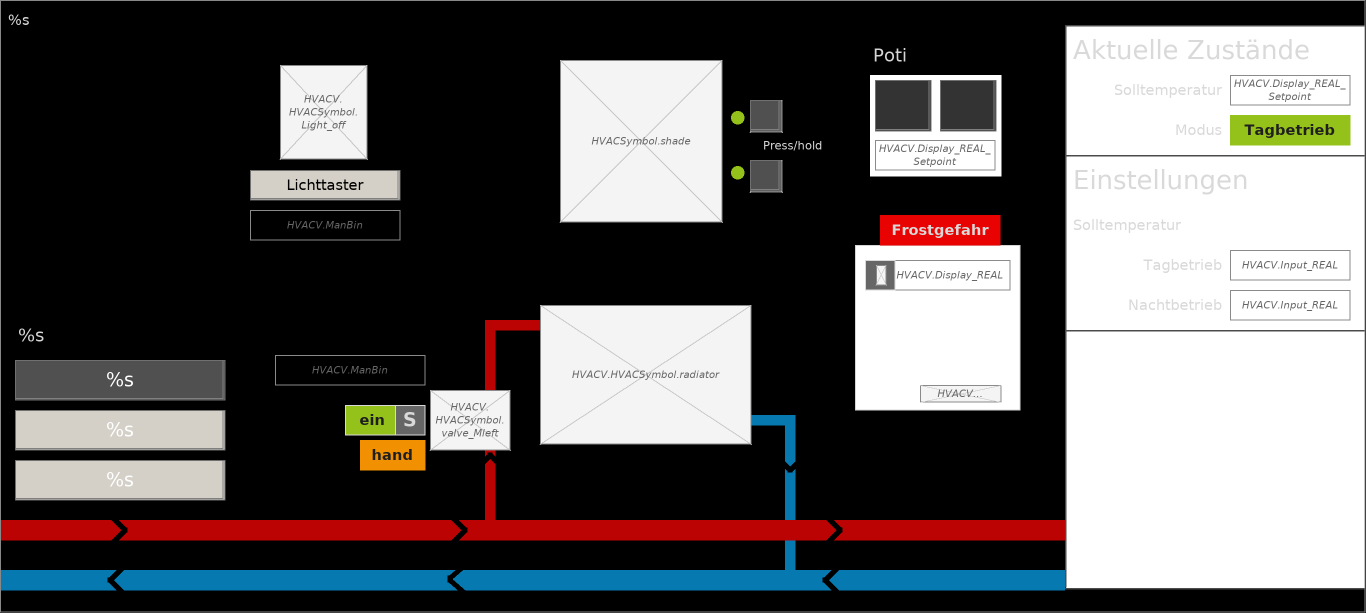
VISUALIZATION Zone_F_Therm_Start  // 1366x613
VAR_IN_OUT
	FB : Zone_F_Therm;
	
END_VAR
    Rectangle (870,75 131x101)
    Rectangle (485,440 10x90)
    Rectangle (785,415 10x170)
    Rectangle (0,520 1280x20)
    Rectangle (0,570 1280x20)
    Polyline (840,565) (825,580) (840,595)
    Polyline (825,515) (840,530) (825,545)
    Polyline (475,470) (490,455) (505,470)
    Polyline (775,455) (790,470) (805,455)
    Polyline (125,565) (110,580) (125,595)
    Polyline (110,515) (125,530) (110,545)
    Polyline (465,565) (450,578) (450,580) (465,593) (465,593) (465,595)
    Polyline (450,515) (465,530) (450,545)
    Rectangle (740,415 50x10)
    Rectangle (485,320 56x10)
    Rectangle (485,320 10x80)
    Image (430,390 80x60), image: HVACV.HVACSymbol.valve_Mleft
    Rectangle (1065,25 300x565)
    Rectangle (1065,155 300x1)
    Rectangle (1070,30 290x40), "Aktuelle Zustände"
    Rectangle (1075,75 150x30), "Solltemperatur"
    Rectangle (1075,115 150x30), "Modus"
    RoundedRectangle (1230,115 120x30), "Nachtbetrieb"
    RoundedRectangle (1230,115 120x30), "Tagbetrieb", invisible if: NOT FB.MODUS
    Rectangle (1065,25 300x1)
    Rectangle (1065,330 300x1)
    Rectangle (1070,160 290x40), "Einstellungen"
    Rectangle (1075,250 150x30), "Tagbetrieb"
    Rectangle (1075,290 150x30), "Nachtbetrieb"
    Rectangle (1070,205 170x40), "Solltemperatur"
    Rectangle (1065,25 1x562)
    Rectangle (1065,588 300x1)
    Rectangle (5,0 970x40), "%s", text variable: FB.Zeile1
    Line (325,495)
    RoundedRectangle (360,440 65x30), "hand", invisible if: FB.VEN.eAOO=0
    Image (540,305 211x139), image: HVACV.HVACSymbol.radiator
    RoundedRectangle (855,245 165x165)
    Image (920,385 81x17), image: HVACV.HVACImage.HVAC_Logo
    Rectangle (855,225 160x20), "Raumbediengerät"
    RoundedRectangle (880,215 120x30), "Frostgefahr", invisible if: NOT FB.FROST
    RoundedRectangle (345,405 55x30), "aus"
    RoundedRectangle (345,405 55x30), "ein", invisible if: NOT FB.VEN.xHB
    Frame (890,260 120x30)
        shows HVACV.Display_REAL(rValue := FB.RBG_TF_RT, bDecimals := 1, xAlarm := FB.RBG_TF_RT_STO, sUnit := '°C')
    RoundedRectangle (395,405 30x30), "S"
    RoundedRectangle (865,260 30x30)
    Image (876,265 10x20), image: HVACV.HVACImage.thermometer1
    Frame (275,355 150x30)
        shows HVACV.ManBin(eManModeB := FB.VEN.eManModeB)
    Frame (1230,75 120x30)
        shows HVACV.Display_REAL_Setpoint(rSetpoint := FB.SOLLTEMP, bDecimals := 1, sUnit := '°C')
    Frame (1230,250 120x30)
        shows HVACV.Input_REAL(rValue := FB.SOLLW_TAG.rSetPoint, bDecimals := 1, sUnit := '°C', rMinInputVisu := 10, rMaxInputVisu := 35, sDialogTitle := 'Solltemperatur Tagbetrieb')
    Frame (1230,290 120x30)
        shows HVACV.Input_REAL(rValue := FB.SOLLW_NACHT.rSetPoint, bDecimals := 1, sUnit := '°C', rMinInputVisu := 10, rMaxInputVisu := 35, sDialogTitle := 'Solltemperatur Tagbetrieb')
    Frame (875,140 120x30)
        shows HVACV.Display_REAL_Setpoint(rSetpoint := PRG.Room_1.VisuPoti.rOut, bDecimals := 1, sUnit := 'K')
    Rectangle (940,80 55x51)
    Rectangle (945,85 46x44), "+"
    Rectangle (875,80 55x51)
    Rectangle (880,80 46x44), "-"
    Button (875,80 56x51)
        OnMouseClick:  ToggleVariable=PRG.Room_1.VisuPoti.xButtonDown
    Button (940,80 56x51)
        OnMouseClick:  ToggleVariable=PRG.Room_1.VisuPoti.xButtonUp
    Button (15,360 210x40), "%s", text variable: FB.AS.sTitleM0, colour toggle: FB.AS.eMode = 0
        OnMouseClick: execute { FB.AS.eMode := 0; }
    Button (15,410 210x40), "%s", text variable: FB.AS.sTitleM1, colour toggle: FB.AS.eMode =1
        OnMouseClick: execute { FB.AS.eMode := 1; }
    Button (15,460 210x40), "%s", text variable: FB.AS.sTitleM2, colour toggle: FB.AS.eMode =2
        OnMouseClick: execute { FB.AS.eMode := 2; }
    Rectangle (15,320 216x31), "%s", text variable: FB.AS.sTitle
    Rectangle (870,40 131x31), "Poti"
    Image (560,60 162x162), image: HVACSymbol.shade
    Button (250,170 150x30), "Lichttaster"
        tap FB.Lichttaster_Visu
    Frame (250,210 150x30)
        shows HVACV.ManBin(eManModeB := FB.Light_Man.eManMode)
    Image (750,100 32x32), angle 90, image: HVACImage.arrow_left
    Image (750,160 32x32), angle 270, image: HVACImage.arrow_left
    Ellipse (730,110 15x15), invisible if: NOT FB.JAL_AUF_HB
    Ellipse (730,165 15x15), invisible if: NOT FB.JAL_ZU_HB
    Button (750,100 31x31)
        tap FB.JAL_AUF_VISU
    Button (750,160 31x31)
        tap FB.JAL_AB_VISU
    Image (280,65 87x94), invisible if: NOT FB.Licht_HB, image: HVACV.HVACSymbol.Light_On
    Image (280,65 87x94), invisible if: FB.Licht_HB, image: HVACV.HVACSymbol.Light_off
    Rectangle (760,130 131x31), "Press/hold"
END_VISUALIZATION

// Device/Application/Macros and frames/HeatingCircuit/Valve_Frames/ValveAnalog_Parameter_Dialog
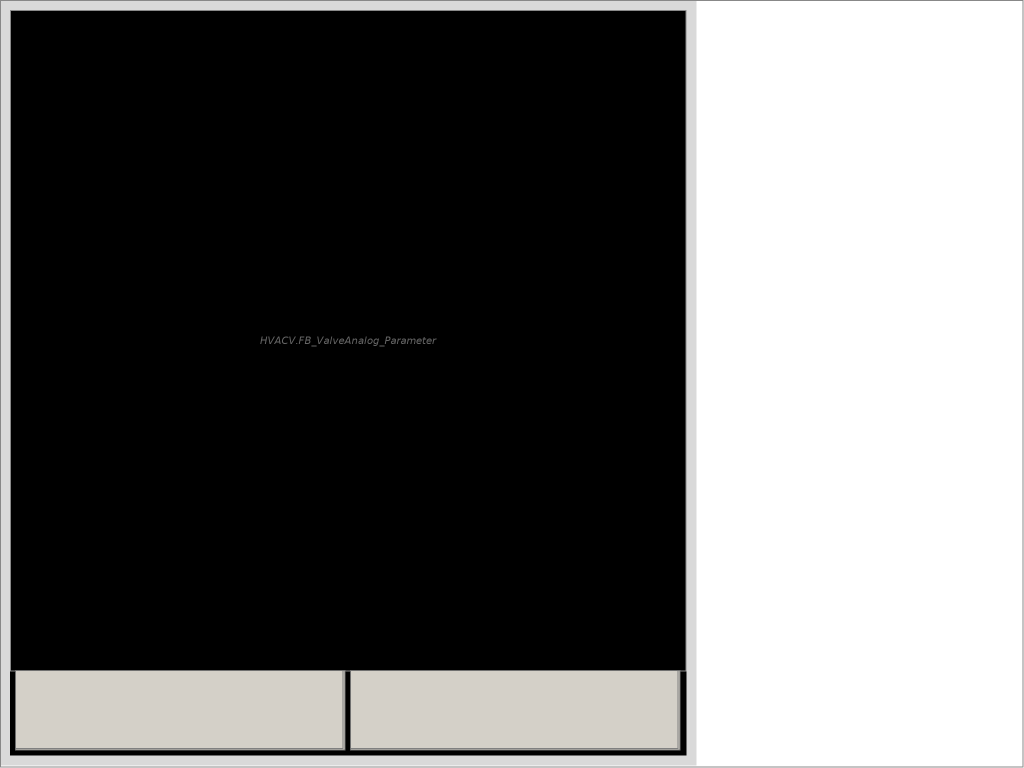
VISUALIZATION ValveAnalog_Parameter_Dialog  // 1024x768
VAR_IN_OUT
	FB_ValveAnalog : HVAC.ValveAnalog;
END_VAR
    Rectangle (0,0 696x765)
    Rectangle (10,10 676x745)
    Frame (10,10 676x661)
        shows HVACV.FB_ValveAnalog_Parameter(FB_ValveAnalog := FB_ValveAnalog)
    Frame (350,670 330x80)
        shows HVACV.OK_Button(iPixel_Right := 30)
    Frame (15,670 330x80)
        shows HVACV.Exit_Button(iPixel_Right := 30)
    Button (350,670 330x80), tooltip "Schließen und Änderung übernehmen."
        OnMouseClick:  Dialog=ValveAnalog_Parameter_Dialog, Result=OK, NumpadKeypadSet=True
    Button (15,670 330x80)
        OnMouseClick:  Dialog=ValveAnalog_Parameter_Dialog, Result=Cancel, NumpadKeypadSet=True
    hotkey  Id=481037385728, Key=KeyDown=True, KeyName=ESCAPE, VisuElemId=264
    hotkey  Id=481038434304, Key=KeyName=ESCAPE, VisuElemId=264
    hotkey  Id=481039482880, Key=KeyDown=True, KeyName=RETURN_KEY, VisuElemId=266
    hotkey  Id=481040531456, Key=KeyName=RETURN_KEY, VisuElemId=266
END_VISUALIZATION

// Device/Application/Visu/3_Settings/Settings_Persistence
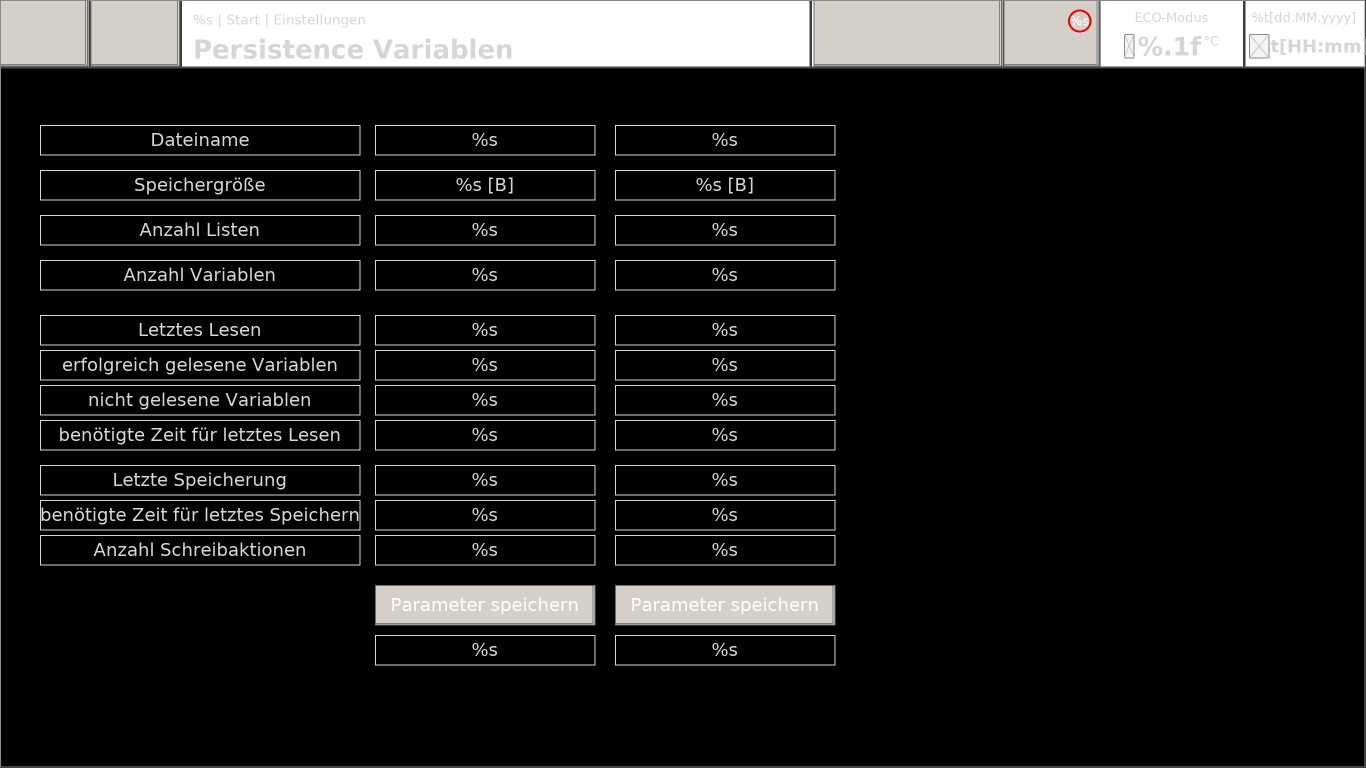
VISUALIZATION Settings_Persistence  // 1366x768
    Rectangle (40,125 320x30), "Dateiname"
    Rectangle (40,170 320x30), "Speichergröße"
    Rectangle (40,215 320x30), "Anzahl Listen"
    Rectangle (40,260 320x30), "Anzahl Variablen"
    Rectangle (40,315 320x30), "Letztes Lesen"
    Rectangle (40,350 320x30), "erfolgreich gelesene Variablen"
    Rectangle (40,385 320x30), "nicht gelesene Variablen"
    Rectangle (40,420 320x30), "benötigte Zeit für letztes Lesen"
    Rectangle (40,465 320x30), "Letzte Speicherung"
    Rectangle (40,500 320x30), "benötigte Zeit für letztes Speichern"
    Rectangle (40,535 320x30), "Anzahl Schreibaktionen"
    Frame (0,0 1366x70)
        shows Header_Frame()
    Rectangle (190,5 545x30), "%s | Start | Einstellungen", text variable: PRG.GebVar
    Rectangle (190,32 545x35), "Persistence Variablen"
    Rectangle (375,125 220x30), "%s", text variable: PersistenceManager.INST_HVAC_Parameter.sChannelName
    Rectangle (375,170 220x30), "%s [B]", text variable: PersistenceManager.INST_HVAC_Parameter.udiDataMemSize
    Rectangle (375,215 220x30), "%s", text variable: PersistenceManager.INST_HVAC_Parameter.uiNumberOfLists
    Rectangle (375,260 220x30), "%s", text variable: PersistenceManager.INST_HVAC_Parameter.udiNumberOfVars
    Rectangle (375,315 220x30), "%s", text variable: PersistenceManager.INST_HVAC_Parameter.dtLastReading
    Rectangle (375,350 220x30), "%s", text variable: PersistenceManager.INST_HVAC_Parameter.udiNumberVarsOk
    Rectangle (375,385 220x30), "%s", text variable: PersistenceManager.INST_HVAC_Parameter.udiNumberVarsNotOk
    Rectangle (375,420 220x30), "%s", text variable: PersistenceManager.INST_HVAC_Parameter.tTimeForReading
    Rectangle (375,465 220x30), "%s", text variable: PersistenceManager.INST_HVAC_Parameter.dtLastSaving
    Rectangle (375,500 220x30), "%s", text variable: PersistenceManager.INST_HVAC_Parameter.tTimeForWriting
    Rectangle (375,535 220x30), "%s", text variable: PersistenceManager.INST_HVAC_Parameter.udiWritingCycles
    Button (375,585 220x40), "Parameter speichern"
        toggle PersistenceManager.INST_HVAC_Parameter.xDoSave
    Rectangle (375,635 220x30), "%s", text variable: PersistenceManager.INST_HVAC_Parameter.xDoSave
    Rectangle (615,125 220x30), "%s", text variable: PersistenceManager.INST_HVAC_Counter.sChannelName
    Rectangle (615,170 220x30), "%s [B]", text variable: PersistenceManager.INST_HVAC_Counter.udiDataMemSize
    Rectangle (615,215 220x30), "%s", text variable: PersistenceManager.INST_HVAC_Counter.uiNumberOfLists
    Rectangle (615,260 220x30), "%s", text variable: PersistenceManager.INST_HVAC_Counter.udiNumberOfVars
    Rectangle (615,315 220x30), "%s", text variable: PersistenceManager.INST_HVAC_Counter.dtLastReading
    Rectangle (615,350 220x30), "%s", text variable: PersistenceManager.INST_HVAC_Counter.udiNumberVarsOk
    Rectangle (615,385 220x30), "%s", text variable: PersistenceManager.INST_HVAC_Counter.udiNumberVarsNotOk
    Rectangle (615,420 220x30), "%s", text variable: PersistenceManager.INST_HVAC_Counter.tTimeForReading
    Rectangle (615,465 220x30), "%s", text variable: PersistenceManager.INST_HVAC_Counter.dtLastSaving
    Rectangle (615,500 220x30), "%s", text variable: PersistenceManager.INST_HVAC_Counter.tTimeForWriting
    Rectangle (615,535 220x30), "%s", text variable: PersistenceManager.INST_HVAC_Counter.udiWritingCycles
    Button (615,585 220x40), "Parameter speichern"
        toggle PersistenceManager.INST_HVAC_Counter.xDoSave
    Rectangle (615,635 220x30), "%s", text variable: PersistenceManager.INST_HVAC_Counter.xDoSave
END_VISUALIZATION

// Device/Application/Visu/1_Objects/HC_1/Settings_HC_1
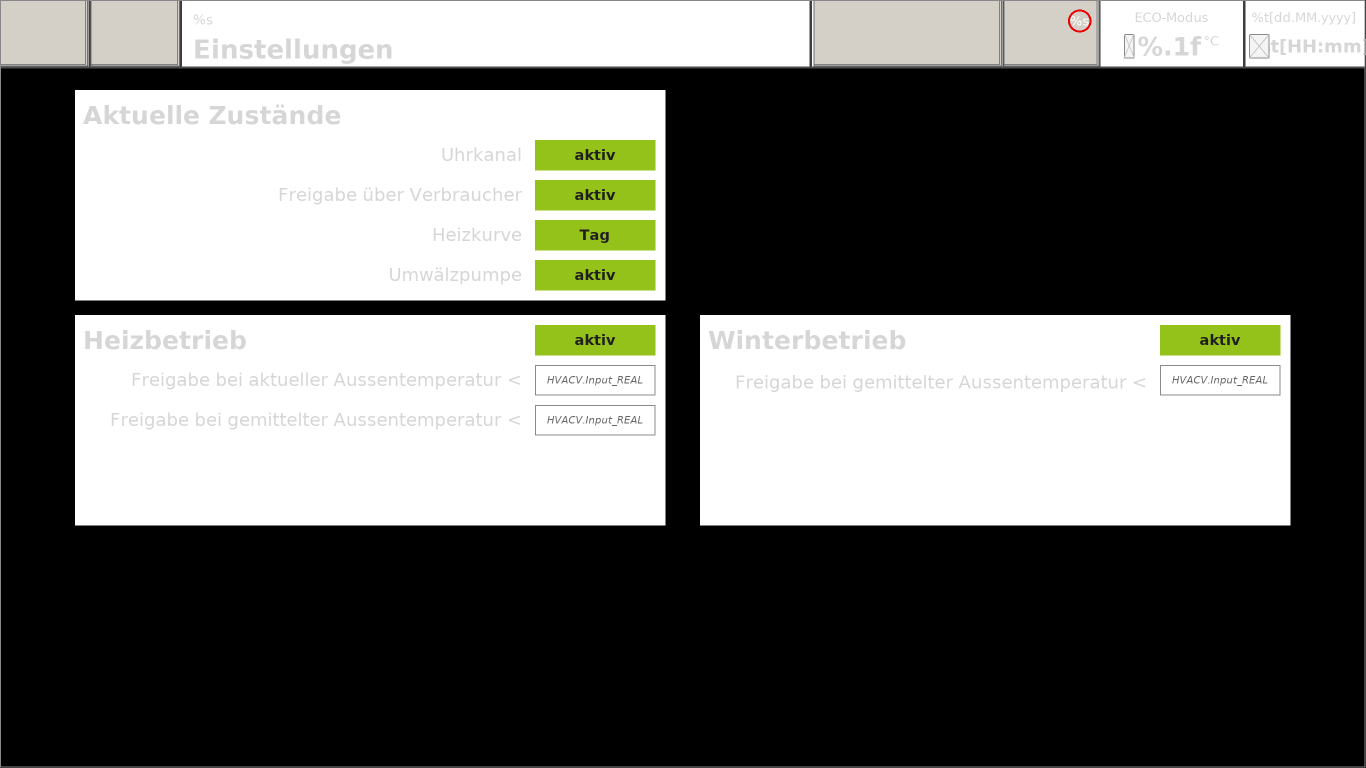
VISUALIZATION Settings_HC_1  // 1366x768
    Frame (0,0 1366x70)
        shows Header_Frame()
    Rectangle (190,5 545x30), "%s", text variable: CONCAT( CONCAT(PRG.GebVar, ' | Start | Objekte | '), Prg.HC_1.Title)
    Rectangle (190,32 545x35), "Einstellungen", text variable: PRG.HC_1.Title
    Frame (0,70 1366x696)
        shows HeatingCircuit_VenA_Settings(FB := PRG.HC_1)
END_VISUALIZATION

// Device/Application/Macros and frames/HeatingCircuit/HeatingCircuit_VenA_Settings
